      L     #LAST_BCD;
      L     #AKT_BCD; // Prüfen ob der BCD
      ==I   ;
      =     #NODIFF; // kein Unterschied in der Anwahl
      T     #LAST_BCD; // seit dem letzten Programmzyklus
NETWORK
TITLE =Verzögerungszeit BCD-WERT-Änderung bis zur Ausgangsumschaltung

      U     #DIFF;
      U     #NODIFF;
      =     L      1.0;
      BLD   103;
      CALL #TON (
           IN                       := L      1.0,
           PT                       := #DELAY,
           Q                        := #QT);

      NOP   0;
NETWORK
TITLE =

      U     #DIFF; // Wert wurde verändert
      U     #QT; // Wartezeit für Umschaltung abgelaufen
      SAVE  ; // Umschaltereignis auf ENO-AUSGANG
      SPB   SAVE; // neue Werte speichern
      BEA   ;

SAVE: L     #AKT_BCD; // Aktuelle BCD-Zahl
      T     #LAST_BCD_AKTIV; // als letzte Zahl speichern

      L     #AKT_BCD; // Aktuelle BCD-Zahl = Bit-Nr im Ausgangs-WORD
      L     1; // Eine 1 um Anzahl "BCD-Zahl" nach links schieben
      SLW   ;
      TAW   ; // Low- und High- Byte im WORD tauschen
      T     DIW [AR2,P#6.0]; // Wert an Ausgänge schreiben (Q1 bis Q9)

END_FUNCTION_BLOCK

FUNCTION_BLOCK "UP_DOWN_INT"
TITLE =UP_DOWN_INT: Wert mit Tasten vergrößeren und verkleinern
//AUTOR: Stefan Maag, Dipl.-Ing. (FH) Elektrotechnik
//DATUM: 1/2005
//
//AENDERUNGSVERMERKE:
//--------------------------------------------------------------------------------
//DATUM        NAME            AENDERUNG
//--------------------------------------------------------------------------------
//
//--------------------------------------------------------------------------------
//
//HINWEISE:
AUTHOR : 'S.Maag'
VERSION : 0.1


VAR_INPUT
  UP : BOOL ;
  DOWN : BOOL ;
  SET : BOOL ;
  SET_VALUE : INT ;
  MIN : INT ;
  MAX : INT ;
  STEP_SLOW : INT ;
  STEP_FAST : INT ;
  STEP_PULS : INT ;
  TAKT : TIME ;
  DELAY_FAST : TIME ;	//Verzögerungszeit für Umschalten auf Schnell
END_VAR
VAR_IN_OUT
  VALUE : INT ;
END_VAR
VAR
  lb_FP_UP : BOOL ;
  lb_FP_DOWN : BOOL ;
  UP_PULS : BOOL ;
  DOWN_PULS : BOOL ;
  FAST : BOOL ;
  TAKT_PULS : BOOL ;
  T1 : "TON";
  T2 : "TON";
END_VAR
BEGIN
NETWORK
TITLE =
//23.06.2012 Slow daktiviert


NETWORK
TITLE =Puls UP
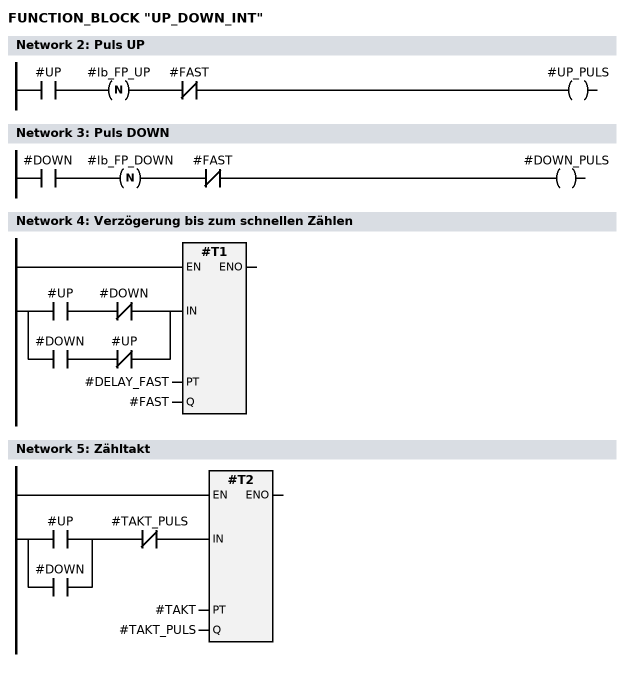

      U     #UP;
      FN    #lb_FP_UP;
      UN    #FAST;
      =     #UP_PULS;
NETWORK
TITLE =Puls DOWN

      U     #DOWN;
      FN    #lb_FP_DOWN;
      UN    #FAST;
      =     #DOWN_PULS;
NETWORK
TITLE =Verzögerung bis zum schnellen Zählen

      U(    ;
      U     #UP;
      UN    #DOWN;
      O     ;
      U     #DOWN;
      UN    #UP;
      )     ;
      =     L      0.0;
      BLD   103;
      CALL #T1 (
           IN                       := L      0.0,
           PT                       := #DELAY_FAST,
           Q                        := #FAST);

      NOP   0;
NETWORK
TITLE =Zähltakt

      U(    ;
      O     #UP;
      O     #DOWN;
      )     ;
      UN    #TAKT_PULS;
      =     L      0.0;
      BLD   103;
      CALL #T2 (
           IN                       := L      0.0,
           PT                       := #TAKT,
           Q                        := #TAKT_PULS);

      NOP   0;
NETWORK
TITLE =SET: Wert setzen

      UN    #SET;
      SPB   NE5;
      L     #SET_VALUE;
      SPA   CHK;
NE5:  NOP   0;

NETWORK
TITLE =
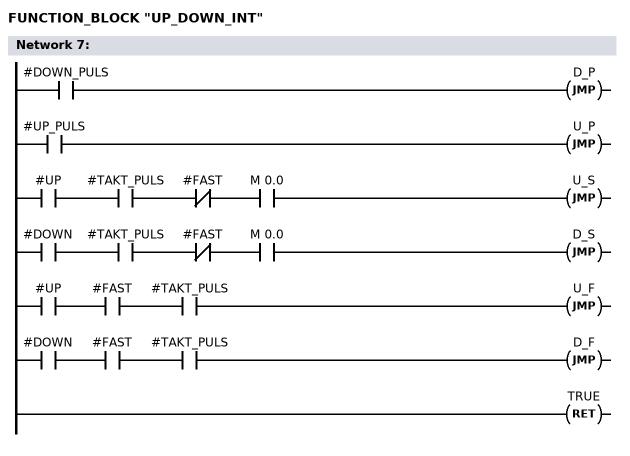

      U     #DOWN_PULS;
      SPB   D_P;

      U     #UP_PULS;
      SPB   U_P;

      U     #UP;
      U     #TAKT_PULS;
      UN    #FAST;
      U     M      0.0;
      SPB   U_S;

      U     #DOWN;
      U     #TAKT_PULS;
      UN    #FAST;
      U     M      0.0;
      SPB   D_S;

      U     #UP;
      U     #FAST;
      U     #TAKT_PULS;
      SPB   U_F;

      U     #DOWN;
      U     #FAST;
      U     #TAKT_PULS;
      SPB   D_F;
      BEA   ;

NETWORK
TITLE =

U_S:  NOP   0; // Up slow
      L     #VALUE;
      L     #STEP_SLOW;
      +I    ;
      SPA   CHK;

U_F:  NOP   0; // Up fast
      L     #VALUE;
      L     #STEP_FAST;
      +I    ;
      SPA   CHK;

U_P:  NOP   0; // Up pulse
      L     #VALUE;
      L     #STEP_PULS;
      +I    ;
      SPA   CHK;


D_S:  NOP   0; // Down slow
      L     #VALUE;
      L     #STEP_SLOW;
      -I    ;
      SPA   CHK;

D_P:  NOP   0; // Down puls
      L     #VALUE;
      L     #STEP_PULS;
      -I    ;
      SPA   CHK;

D_F:  NOP   0; // Down fast
      L     #VALUE;
      L     #STEP_FAST;
      -I    ;

CHK:  L     #MIN; // Wert auf Min/Max begrenzen
      <I    ;
      SPB   SAVE;
      TAK   ;
      L     #MAX;
      >I    ;
      SPB   SAVE;
      TAK   ;
SAVE: T     #VALUE;

END_FUNCTION_BLOCK

FUNCTION_BLOCK "m7b_SchuetzUeberwachung"
TITLE =Schützfehlerüberwachung mit Rückmeldekontakt
//AUTOR: Stefan Maag, Dipl.-Ing. (FH) Elektrotechnik
//DATUM: 12/2009
//INTERNET: www.maagic7.de
//
//AENDERUNGSVERMERKE:
//--------------------------------------------------------------------------------
//DATUM        NAME            AENDERUNG
//--------------------------------------------------------------------------------
//
//--------------------------------------------------------------------------------
//
//HINWEISE:
AUTHOR : 'S.Maag'
FAMILY : Maagic7
VERSION : 0.1


VAR_INPUT
  K : BOOL ;
  RM : BOOL ;
  IEC_TIME : TIME ;
END_VAR
VAR
  MI_TON : "TON";
END_VAR
VAR_TEMP
  XOR_RESULT : BOOL ;
  Q_TON : BOOL ;
END_VAR
BEGIN
NETWORK
TITLE =Schütz <> Rückmdlung ?

      X     #K;
      X     #RM;
      =     #XOR_RESULT;

NETWORK
TITLE =Zeitverzögerung, wenn Ansteuerung <> Rückmeldung



      U     #XOR_RESULT;
      =     L      1.0;
      BLD   103;
      CALL #MI_TON (
           IN                       := L      1.0,
           PT                       := #IEC_TIME,
           Q                        := #Q_TON);

      NOP   0;
NETWORK
TITLE =ENO-Ausgang : Fehlerausgang

      U     #Q_TON;
      SAVE  ;
      CLR   ;

END_FUNCTION_BLOCK

FUNCTION_BLOCK "POSI"
TITLE =Positionierung Achse mit Delay für Nachpositionierung bzw. Ready
//Positionierung Achse als Schrittsteuerung:
//
//Lageregelung nur während der timDelayReady.
//Soll ohne die Möglichkeit der Nachpositionierung sofort bei erreichen der
//Stopdifferenz fest abgeschaltet werden, dann timDelayReady =0
//
//
//[IN]
//FRG :       Freigabe, wenn Low, dann Abbruch der Positionierung
//SOLL:       Sollposition Achse
//IST :       Istposition Achse
//STOP_DIFF:  Vorabschaltentfernung
//TOL_POS_OK: Toleranz für Position ok Prüfung
//timDelayReady : Verzögerung für Ready (Nachpositionierung nur in dieser Zeit)
//
//[IN_OUT]
//START:      Befehl Positionierung Start, wird bei Ende oder Abbruch gelöscht
//
//[OUT]
//PLUS:       Fahrtrichtung Plus (vorw.)
//MINUS:      Fahrtrichtung Minus (rückw.)
//READY:      Positionierablauf korrekt beendet
//POS_OK:     Position innerhalb der Toleranz (ständige Prüfung)
//DSP_SNR:    Schrittnummer Positionierablauf
//
//FC_ENO:     zeigt an, dass Positionierung läuft
//
//AUTOR: Stefan Maag, Dipl.-Ing. (FH) Elektrotechnik
//DATUM: 9/2007
//
//AENDERUNGSVERMERKE:
//--------------------------------------------------------------------------------
//DATUM        NAME        AENDERUNG
//--------------------------------------------------------------------------------
//20.11.2017   S.Maag     Nachpositionierung eingeführt.
//                        timDelayReady gibt, an wie lange der Antrieb in
//                        korrekter Position sein muss, bis READY ausgegeben
//                        wird. Dann wird nicht mehr nachpositioniert.
//                        Dies ist insbesondere bei etwas instabilen Positons-
//                        erfassungen wie Laser Entfernungsmesser nötig. Sonst
//                        kann es sein, dass der Laser etwas wackelt, es wird
//                        gestoppt, die Position ist jedoch nicht im Fenster.
//--------------------------------------------------------------------------------
//
//HINWEISE:
AUTHOR : 'S.Maag'
VERSION : 0.1


VAR_INPUT
  FRG : BOOL ;	//Freigabe
  SOLL : DINT ;	//Sollwert
  IST : DINT ;	//Istwert Achse
  STOP_DIFF : DINT ;	//Vorabschaltpunkt
  TOL_POS : DINT ;	//Toleranz für Positionierung
  TOL_POS_OK : DINT ;	//Toleranz für Position ok Meldung
  timDelayReady : TIME ;
END_VAR
VAR_OUTPUT
  PLUS : BOOL ;	//Fahrtrichtung PLUS
  MINUS : BOOL ;	//Fahrtrichtung MINUS
  READY : BOOL ;	//Positionierung fertig
  POS_OK : BOOL ;	//Position innerhalb Toleranz ok
  DSP_SNR : INT ;	//Schrittnummer Positionierung, STATE
END_VAR
VAR_IN_OUT
  START : BOOL ;
END_VAR
VAR
  SNR : INT ;
  POS_DIFF : DINT ;	//aktuelle Positionsdifferenz
  FRG_GO : BOOL ;
  POS_INTERVAL : BOOL ;
  Q_TON_FRG_GO_OFF : BOOL ;
  mi_TON_FRG_GO_OFF : "TON";
END_VAR
VAR_TEMP
  tmpPosDIFF : DINT ;
  tmp_timDelay : TIME ;
END_VAR
BEGIN
NETWORK
TITLE =



NETWORK
TITLE =Zeit mindestens 1ms (da 0=RESET für IEC-Timer)

      L     L#1;
      L     #timDelayReady;
      UC    FC    21;
      T     #tmp_timDelay;

NETWORK
TITLE =Zeit Freiagbe GO ist AUS (Achse ist positioniert)

      UN    #FRG_GO;
      =     L      8.0;
      BLD   103;
      CALL #mi_TON_FRG_GO_OFF (
           IN                       := L      8.0,
           PT                       := #tmp_timDelay,
           Q                        := #Q_TON_FRG_GO_OFF);

      NOP   0;
NETWORK
TITLE =Signale Fahrtrichtung

      U(    ;
      L     #SOLL;
      L     #IST;
      -D    ;
      T     #POS_DIFF;
      UN    OV;
      SAVE  ;
      CLR   ;
      U     BIE;
      )     ;
      U     #FRG_GO;
      UN    #POS_INTERVAL;
      =     L      8.0;
      U     L      8.0;
      U     >0;
      =     #PLUS;
      U     L      8.0;
      U     <0;
      =     #MINUS;
NETWORK
TITLE =Toleranzprüfung Position

      U(    ;
      L     #POS_DIFF;
      L     L#0;
      <D    ;
      )     ;
      SPBNB _001;
      L     #POS_DIFF;
      NEGD  ;
      T     #POS_DIFF;
_001: NOP   0;
NETWORK
TITLE =Toleranzprüfung Position
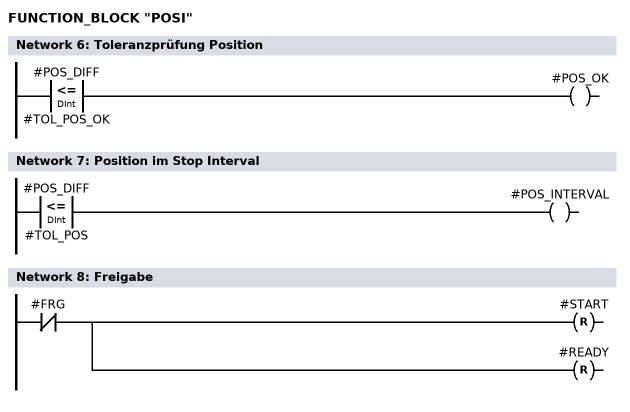

      L     #POS_DIFF;
      L     #TOL_POS_OK;
      <=D   ;
      =     #POS_OK;
NETWORK
TITLE =Position im Stop Interval

      L     #POS_DIFF;
      L     #TOL_POS;
      <=D   ;
      =     #POS_INTERVAL;
NETWORK
TITLE =Freigabe

      UN    #FRG;
      R     #START;
      R     #READY;

NETWORK
TITLE =Standard Ablaufsteuerung mit INIT und CLR-Zweig

      L     #SNR; // Schrittnummer
      SPL   CLR; // Sprungziel bei SNR>max
      SPA   INIT; // 0-Schritt, Initialisierung
      SPA   S1; // Startschritt
      SPA   S2;

CLR:  SET   ; // CLR
// hier die bei CLR zu löschenden Merker eintragen
      R     #START;
      R     #FRG_GO;

      L     1; // Schrittnummer
      T     #SNR; // auf Startschritt stellen
      T     #DSP_SNR; // Schrittnummer Anzeige
      SPA   END;

INIT: SET   ; // Initalisierung
      CLR   ;
      SPA   CLR;
      SPA   SET; // wird nur benötigt, damit die Entwicklungsumgebung die Sprungmarke nicht löscht

NETWORK
TITLE =Schrittweiterschaltung, bzw. Bausteinende

NEXT: L     #SNR; // NEXT : Schrittnummer auf nächsten
      +     1; // Schritt
SET:  T     #SNR; // Schritt setzten

END:  L     #SNR; // Sprungmarke für Baustein ENDE
      T     #DSP_SNR; // Schrittnummer Anzeige
      L     1; // Wenn Ablauf läuft, dann ENO-Ausgang = 1
      >I    ;
      SAVE  ;
      CLR   ;
      BEA   ;

NETWORK
TITLE =Positionierung START?
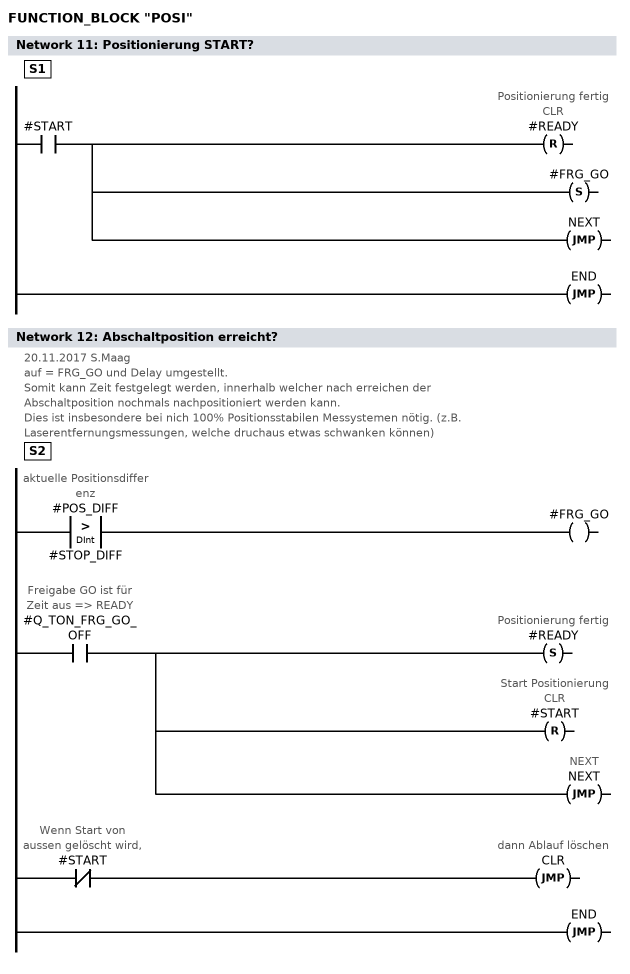

S1:   U     #START;
      R     #READY; // Positionierung fertig CLR
      S     #FRG_GO;
      SPB   NEXT;
      SPA   END;

NETWORK
TITLE =Abschaltposition erreicht?
//20.11.2017 S.Maag
//auf = FRG_GO und Delay umgestellt.
//Somit kann Zeit festgelegt werden, innerhalb welcher nach erreichen der
//Abschaltposition nochmals nachpositioniert werden kann.
//Dies ist insbesondere bei nich 100% Positionsstabilen Messystemen nötig. (z.B.
//Laserentfernungsmessungen, welche druchaus etwas schwanken können)
S2:   NOP   0;
      L     #POS_DIFF; // aktuelle Positionsdifferenz
      L     #STOP_DIFF; // Vorabschaltpunkt
      >D    ;
      =     #FRG_GO;

      U     #Q_TON_FRG_GO_OFF; // Freigabe GO ist für Zeit aus => READY
      S     #READY; // Positionierung fertig
      R     #START; // Start Positionierung CLR
      SPB   NEXT; // NEXT

      UN    #START; // Wenn Start von aussen gelöscht wird,
      SPB   CLR; // dann Ablauf löschen
      SPA   END;


END_FUNCTION_BLOCK

FUNCTION_BLOCK "m7b_FU_RFR"
TITLE =Reglerfreigabe mit Nachlauf aus vw/rw Signal erzeugen
//AUTOR: Stefan Maag, Dipl.-Ing. (FH) Elektrotechnik
//DATUM: 01/2013
//INTERNET: www.maagic7.de
//
//AENDERUNGSVERMERKE:
//--------------------------------------------------------------------------------
//DATUM        NAME         AENDERUNG
//--------------------------------------------------------------------------------
//13.06.2020   S.Maag       in Library aufgenommen
//--------------------------------------------------------------------------------
//
//HINWEISE:
AUTHOR : 'S.Maag'
VERSION : 0.1


VAR_INPUT
  vw : BOOL ;	//vorwärts
  rw : BOOL ;	//rückwärts
  FRG : BOOL ;
  timTON_MSG : TIME ;	//Verzögerung Meldung RFR
  timTOF_RFR : TIME ;	//Nachlauf Reglerfreigabe
END_VAR
VAR_OUTPUT
  RFR : BOOL ;	//Ausgang Reglerfreigabe FU
  MSG_RFR : BOOL ;	//Meldung verzögert Reglerfreigabe o.k.
END_VAR
VAR
  Q_TON_MSG : BOOL ;
  Q_TOF_RFR : BOOL ;
  TOF_RFR : "TOF";
  TON_MSG : "TON";
END_VAR
VAR_TEMP
  xTON_MSG_IS_ZERO : BOOL ;
  xTOF_RFR_IS_ZERO : BOOL ;
END_VAR
BEGIN
NETWORK
TITLE =



NETWORK
TITLE =Verzögerungszeit Meldung ist 0 ms
//bei 0ms starten IEC Timer nicht und Ausgang bleibt immer lo,
//Aufruf mit 0ms ist RESET
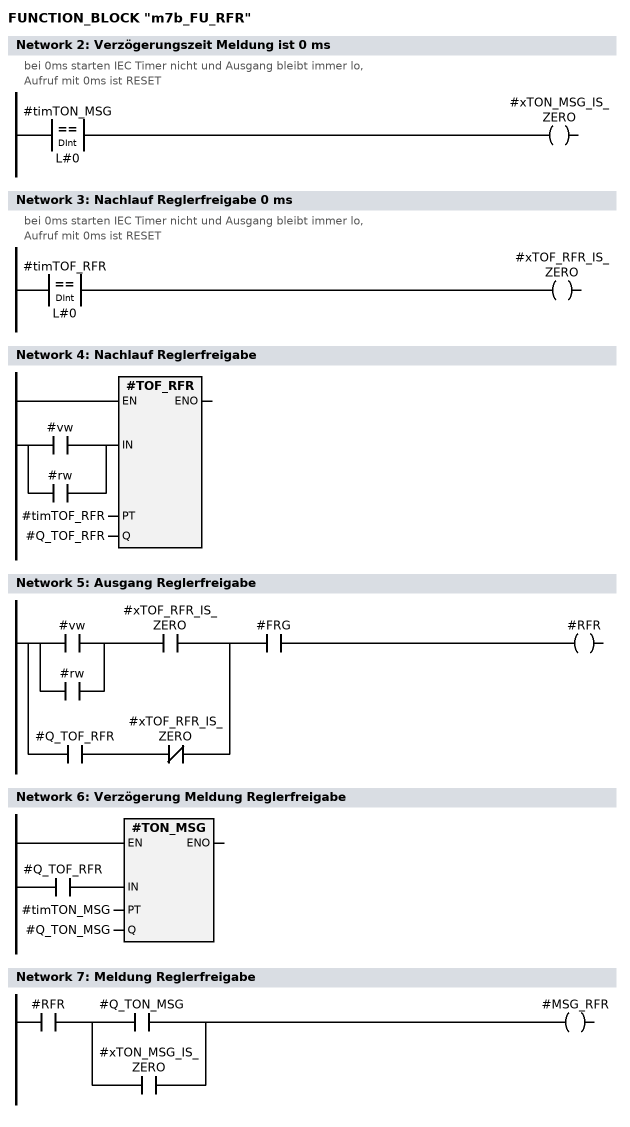
      L     #timTON_MSG;
      L     L#0;
      ==D   ;
      =     #xTON_MSG_IS_ZERO;
NETWORK
TITLE =Nachlauf Reglerfreigabe 0 ms
//bei 0ms starten IEC Timer nicht und Ausgang bleibt immer lo,
//Aufruf mit 0ms ist RESET
      L     #timTOF_RFR;
      L     L#0;
      ==D   ;
      =     #xTOF_RFR_IS_ZERO;
NETWORK
TITLE =Nachlauf Reglerfreigabe

      U(    ;
      O     #vw;
      O     #rw;
      )     ;
      =     L      1.0;
      BLD   103;
      CALL #TOF_RFR (
           IN                       := L      1.0,
           PT                       := #timTOF_RFR,
           Q                        := #Q_TOF_RFR);

      NOP   0;
NETWORK
TITLE =Ausgang Reglerfreigabe

      U(    ;
      U(    ;
      O     #vw;
      O     #rw;
      )     ;
      U     #xTOF_RFR_IS_ZERO;
      O     ;
      U     #Q_TOF_RFR;
      UN    #xTOF_RFR_IS_ZERO;
      )     ;
      U     #FRG;
      =     #RFR;
NETWORK
TITLE =Verzögerung Meldung Reglerfreigabe



      U     #Q_TOF_RFR;
      =     L      1.0;
      BLD   103;
      CALL #TON_MSG (
           IN                       := L      1.0,
           PT                       := #timTON_MSG,
           Q                        := #Q_TON_MSG);

      NOP   0;
NETWORK
TITLE =Meldung Reglerfreigabe

      U     #RFR;
      U(    ;
      O     #Q_TON_MSG;
      O     #xTON_MSG_IS_ZERO;
      )     ;
      =     #MSG_RFR;
END_FUNCTION_BLOCK

FUNCTION_BLOCK "m7b_HydraulicPump"
TITLE =Steuerung Hydraulik mit Lastventil : Hydraulic with load valve
//Steuerung Hydraulikpumpe mit Lastventil!
//
//Einstellbare Nachlaufzeit für Hydraulikpumpe.
//Durch einstellbare Vor- und Nachlaufzeit für Lastventil (Meldung Druck auf
//Hydraulik), verwendbar auch für Hydrauliken mit Porportionalventilen. Bei
//Proportinalsteuerung muss das Lastventil mindestens so lange nachlaufen, wie
//die
//längste Rampenzeit der Ventile. Durch die Vorlaufzeit des Lastventils kann man
//sicherstellen, dass auf jeden Fall Druck ansteht, bevor man die
//Proportionalventile ansteuert.
//
//[IN]
//START        : Befehl, Hydraulik starten
//FRG          : Freigabe für Hydraulik (Netz_ok, Motorschutz usw. verschalten)
//T_HYDR_OFF   : Nachlaufzeit Hydraulikpumpe IEC-Time-Format
//T_Y_LOAD_OFF : Nachlaufzeit Lastventil (> max. Rampenzeiten bei Prop.Ventilen)
//T_MSG_LOAD_ON: Verzögerung Meldung Lastventil ein (Vorlauf Lastventil)
//
//[OUT]
//PUMP          : Ausgang Hydraulikpumpe EIN
//Y_LOAD        : Ausgang Lastventil
//MSG_PUMP_READY: Meldung Hydraulik bereit (=durchgeschleiftes Singal FRG)
//MSG_PUMP_RUN  : Meldung Hydraulikpumpe läuft (fix verzögert 500ms)
//MSG_LOAD_ON   : Meldung Lastventil ist ein (Druck auf Hydraulik) - verzögert
//
//AUTOR: Stefan Maag, Dipl.-Ing. (FH) Elektrotechnik
//DATUM: 11/2008
//INTERNET: www.maagic7.de
//
//AENDERUNGSVERMERKE:
//--------------------------------------------------------------------------------
//DATUM        NAME            AENDERUNG
//--------------------------------------------------------------------------------
//17.09.2010  S.Maag      Reset der iecZeit TOF_HydrPump über 0 im den Zeitwert
//                        damit läuft Pumpe nach Freigabeverlust nicht wieder an
//--------------------------------------------------------------------------------
//
//HINWEISE:
AUTHOR : 'S.Maag'
FAMILY : Maagic7
VERSION : 0.1


VAR_INPUT
  START : BOOL ;	//Hydraulik START
  FRG : BOOL ;	//Freigabe Hydraulikpumpe
  T_HYDR_OFF : TIME ;	//Nachlaufzeit Hydraulikpumpe
  T_Y_LOAD_OFF : TIME ;	//Nachlauf Lastventil
  T_MSG_LOAD_ON : TIME ;
END_VAR
VAR_OUTPUT
  PUMP : BOOL ;	//Ausgang Hydraulikpumpe EIN
  Y_LOAD : BOOL ;	//Ausgang Lastventil
  MSG_PUMP_READY : BOOL ;	//Meldung Hydraulik bereit
  MSG_PUMP_RUN : BOOL ;	//Meldung Hydraulik läuft
  MSG_LOAD_ON : BOOL ;	//Meldung Lastventil ein
END_VAR
VAR
  Q_T_Hydraulic : BOOL ;
  Q_PUMP : BOOL ;
  Q_LOAD_REQ : BOOL ;
  Q_T_LOAD : BOOL ;
  Q_LOAD : BOOL ;
  TOF_HydrPump : "TOF";
  TON_MSG_RUN : "TON";
  TON_LOAD_ON : "TON";
  TOF_LOAD : "TOF";
END_VAR
VAR_TEMP
  DSP_TIME : TIME ;
  m_T_HYDR_OFF : TIME ;
END_VAR
BEGIN
NETWORK
TITLE =



NETWORK
TITLE =Zeit Hydraulik aus auf temporären Zwischenspeicher
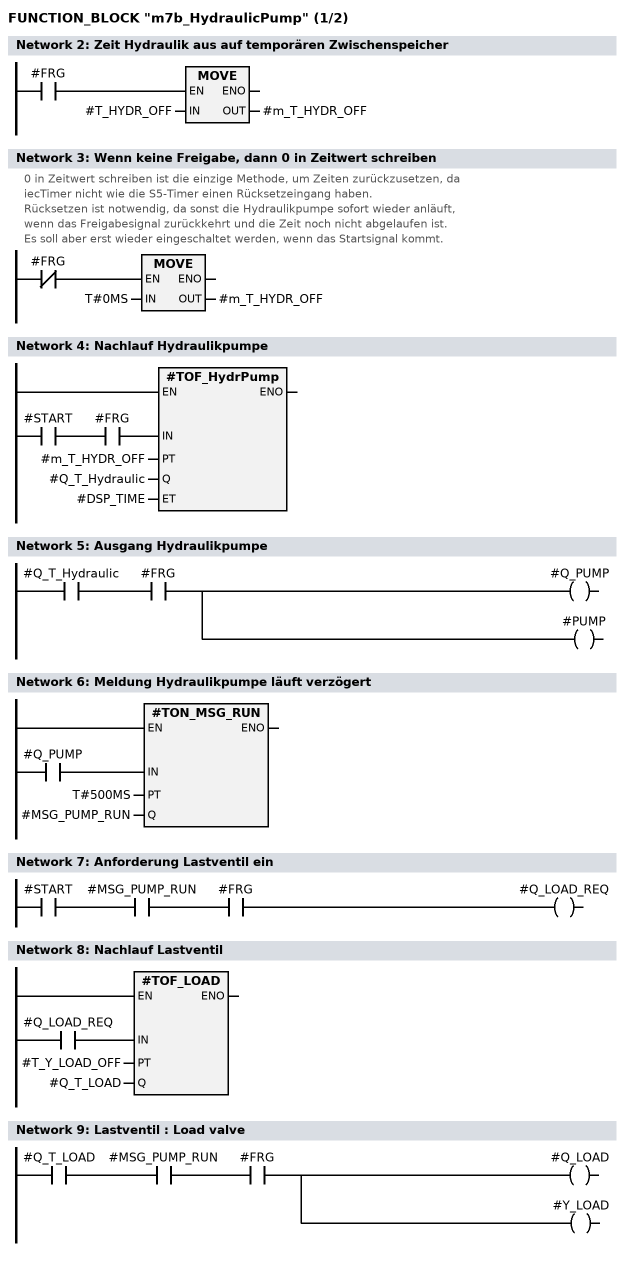

      U     #FRG;
      SPBNB _001;
      L     #T_HYDR_OFF;
      T     #m_T_HYDR_OFF;
_001: NOP   0;
NETWORK
TITLE =Wenn keine Freigabe, dann 0 in Zeitwert schreiben
//0 in Zeitwert schreiben ist die einzige Methode, um Zeiten zurückzusetzen, da
//iecTimer nicht wie die S5-Timer einen Rücksetzeingang haben.
//
//Rücksetzen ist notwendig, da sonst die Hydraulikpumpe sofort wieder anläuft,
//wenn das Freigabesignal zurückkehrt und die Zeit noch nicht abgelaufen ist.
//Es soll aber erst wieder eingeschaltet werden, wenn das Startsignal kommt.
//
      UN    #FRG;
      SPBNB _002;
      L     T#0MS;
      T     #m_T_HYDR_OFF;
_002: NOP   0;
NETWORK
TITLE =Nachlauf Hydraulikpumpe



      U     #START;
      U     #FRG;
      =     L      8.0;
      BLD   103;
      CALL #TOF_HydrPump (
           IN                       := L      8.0,
           PT                       := #m_T_HYDR_OFF,
           Q                        := #Q_T_Hydraulic,
           ET                       := #DSP_TIME);
      NOP   0;
NETWORK
TITLE =Ausgang Hydraulikpumpe

      U     #Q_T_Hydraulic;
      U     #FRG;
      =     #Q_PUMP;
      =     #PUMP;
NETWORK
TITLE =Meldung Hydraulikpumpe läuft verzögert

      U     #Q_PUMP;
      =     L      8.0;
      BLD   103;
      CALL #TON_MSG_RUN (
           IN                       := L      8.0,
           PT                       := T#500MS,
           Q                        := #MSG_PUMP_RUN);

      NOP   0;
NETWORK
TITLE =Anforderung Lastventil ein

      U     #START;
      U     #MSG_PUMP_RUN;
      U     #FRG;
      =     #Q_LOAD_REQ;
NETWORK
TITLE =Nachlauf Lastventil

      U     #Q_LOAD_REQ;
      =     L      8.0;
      BLD   103;
      CALL #TOF_LOAD (
           IN                       := L      8.0,
           PT                       := #T_Y_LOAD_OFF,
           Q                        := #Q_T_LOAD);

      NOP   0;
NETWORK
TITLE =Lastventil : Load valve

      U     #Q_T_LOAD;
      U     #MSG_PUMP_RUN;
      U     #FRG;
      =     #Q_LOAD;
      =     #Y_LOAD;
NETWORK
TITLE =Meldung Lastventil ein : Message Load valve on
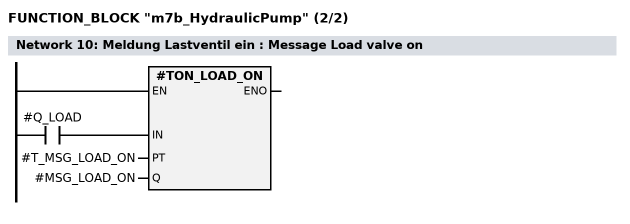

      U     #Q_LOAD;
      =     L      8.0;
      BLD   103;
      CALL #TON_LOAD_ON (
           IN                       := L      8.0,
           PT                       := #T_MSG_LOAD_ON,
           Q                        := #MSG_LOAD_ON);

      NOP   0;
NETWORK
TITLE =ENO-Ausgang = Lastventil

      U     #Q_LOAD;
      SAVE  ;
      CLR   ;

END_FUNCTION_BLOCK

FUNCTION_BLOCK "m7b_ZylSensorCtrl"
TITLE =ZylinderSensorControl, für Zylinder mit 2 Sensoren
//Dier FB erledigt 2 Funktionen
//1. Verzögerung der Zylindersensoren und generieren der Positionsmeldungen
//2. Überwachung der Zylinderbewegungen anhand der max. erlaubten Bewegungszeit
//   bis der entsprechende Positionssensor belegt ist.
//
//Wird in der angebenen Zeit die Zylinderendstellung nicht erreicht, so wird
//ERROR für die entsprechende Richtung ausgegeben. Der ENO-Ausgang des FC erhält
//den ODER-verknüpten Error-Zustand. Ist also bei Fehler, egal welcher Richtung
//High
//
//Auf die SFBs TON, TOF wird verzichtet, da diese bereits je 22Byte an statischen
//Daten verbrauchen. Dies wurde hauptsächlich wegen Speicherproblemen bei den
//kleinen CPUs (312/313) so ausgeführt.
//
//AUTOR: Stefan Maag, Dipl.-Ing. (FH) Elektrotechnik
//DATUM: 3/2008
//INTERNET: www.maagic7.de
//
//HINWEISE: Entstand aus FC7: m7ZylinderFehlerEx
//
//AENDERUNGSVERMERKE:
//--------------------------------------------------------------------------------
//DATUM        NAME            AENDERUNG
//--------------------------------------------------------------------------------
//03/12/2013   S.Maag      SFC64 TimeTick Zeitdifferenz korrigiert
//                         da 31Bit, Fehler bei Überlauf.
//                         UC FC256 "ABS_DIFF_S7SysTime" verwendet
//--------------------------------------------------------------------------------
//
AUTHOR : 'S.Maag'
FAMILY : Maagic7
VERSION : 0.1


VAR_INPUT
  SENS_GST : BOOL ;	//Sensor Grundstellung
  SENS_AST : BOOL ;	//Sensor Arbeitsstellung
  Y_GST : BOOL ;	//Eingang Schaltsignal Grundstellungs-Ventil
  Y_AST : BOOL ;	//Eingang Schaltsignal Arbeitsstellungs-Ventil
  iec_T_Err : TIME ;	//Zeit für Bewegung Fehlerüberwachung, IEC-Format
  iec_T_PosDelay : TIME ;	//Verzögerungszeit für Positionssensoren
END_VAR
VAR_OUTPUT
  POS_GST : BOOL ;	//Position Grundstellung
  POS_AST : BOOL ;	//Position Arbeitsstellung
  ERR_GST : BOOL ;	//Ausgang Fehler Sensor Grundstellung
  ERR_AST : BOOL ;	//Ausgang Fehler Sensor Arbeitsstellung
  STATUS : INT ;	//0=zu 1=auf 2=fährt 3=Fehler zu  4=Fehler auf
END_VAR
VAR
  FP_YGST : BOOL ;	//Flanke positiv Ventil Grundstellung
  FP_YAST : BOOL ;	//Flanke positiv Ventil Arbeitsstellung
  FP_B_GST : BOOL ;
  FP_B_AST : BOOL ;
  aktSysTime : TIME ;
  T_FP_B_GST : TIME ;	//akt. SysZeit Sensor GST Flanke
  T_FP_B_AST : TIME ;	//akt. SysZeit Sensor AST Flanke
  tmpErrTime : TIME ;	//Speichervariable für Zeit
END_VAR
BEGIN
NETWORK
TITLE =aktuelle Systemzeit Zwischenspeichern

      CALL "TIME_TCK" (// aktuelle Systemzeit auslesen
           RET_VAL                  := #aktSysTime);
      NOP   0;
NETWORK
TITLE =Systemzeit bei Sensor Grundstellung belegt
//Zeit bei der Sensor belegt wurde.
      U     #SENS_GST;
      FP    #FP_B_GST;
      SPBNB _001;
      L     #aktSysTime;
      T     #T_FP_B_GST;
_001: NOP   0;
NETWORK
TITLE =Systemzeit bei Sensor Arbeitsstellung belegt
//Zeit bei der Sensor belegt wurde.
      U     #SENS_AST;
      FP    #FP_B_AST;
      SPBNB _002;
      L     #aktSysTime;
      T     #T_FP_B_AST;
_002: NOP   0;
NETWORK
TITLE =Ausgang Position Grundstellung erreicht
//Verzögerung Position Grundstellung
      UN    #SENS_GST; // Sensor Grundstellung nicht aktiv
      R     #POS_GST; // dann Position Grundstellung clr
      SPB   ne4; // Netzwerkende
      L     #aktSysTime; // Wenn Grundstellungssensor High, dann
      L     #T_FP_B_GST; // Zeit überpüfen wie lange bereits
      UC    "m7b_ABS_DIFF_S7SysTime"; // Zeitdifferenz absolut ermitteln
      L     #iec_T_PosDelay; // Wenn größer als Verzögerung,
      >=D   ;
      S     #POS_GST; // dann Position Grundstellung setzen
ne4:  NOP   0;

NETWORK
TITLE =Ausgang Position Arbeitsstellung erreicht
//Verzögerung Position Arbeitsstellung
      UN    #SENS_AST; // Sensor Arbeitsstellung nicht aktiv
      R     #POS_AST; // dann Position Arbeitsstellung clr
      SPB   ne5; // Netzwerkende
      L     #aktSysTime; // Wenn Arbeitsstellungssensor High, dann
      L     #T_FP_B_AST; // Zeit überpüfen wie lange bereits
      UC    "m7b_ABS_DIFF_S7SysTime"; // Zeitdifferenz absolut ermitteln
      L     #iec_T_PosDelay; // Wenn größer als Verzögerung,
      >=D   ;
      S     #POS_AST; // dann Position Arbeitsstellung setzen
ne5:  NOP   0;

NETWORK
TITLE =Zeit bei Bewegung Start speichern

      U     #Y_GST; // falls beide Ventile gleichzeitg angesteuert sind
      U     #Y_AST; // dann Zeitüberwachung solange starten bis ein
      SPB   SVT; // Ventil abgeschaltet wird. Erst dann ist def. Zustand

      U     #Y_GST; // Ventil Grundstellung
      FP    #FP_YGST; // Flanke Ventilansteuerung
      SPB   SVT; // Save Time

      U     #Y_AST; // Ventil Arbeitsstellung
      FP    #FP_YAST; // Flanke Ventilansteuerung
      SPB   SVT; // Save Time

      SPA   NE1;

SVT:  NOP   0; // Zeit bei Bewegung Start speichern
      CALL "TIME_TCK" (// Systemzeit wird zur Bewegungsüberwachung verwendet
           RET_VAL                  := #tmpErrTime);// dadurch erspart man sich Timerübergaben

NE1:  NOP   0;
NETWORK
TITLE =Prüfen, ob beide Sensoren belegt sind => Fehler

      U     #SENS_GST;
      U     #SENS_AST;
      SPBN  NE2;
      =     #ERR_GST;
      =     #ERR_AST;
      SAVE  ;
      BEA   ;
NE2:  NOP   0;

NETWORK
TITLE =Zeit überprüfen, ob Endstellung erreicht ist

      U     #Y_GST; // Ventil Grundstellung
      UN    #SENS_GST; // Sensor GST nicht erreicht
      SPB   TCHK; // Prüfen ob max. Zeit Abgelaufen

      U     #Y_AST; // Ventil Arbeitsstellung
      UN    #SENS_AST; // Sensor Arbeitsstellung nicht erreicht
      SPB   TCHK; // Prüfen ob max. Zeit Abgelaufen

      CLR   ;
      =     #ERR_GST;
      =     #ERR_AST;
      SAVE  ;
      SPA   NE8; // Netzwerkende

TCHK: NOP   0; // Zeit Abgelaufen?
      L     #aktSysTime;
      L     #tmpErrTime; // Zeit bei Start Bewegung
      UC    "m7b_ABS_DIFF_S7SysTime";
      L     #iec_T_Err; // Zeit für Bewegung
      >D    ; // Zeit abgelaufen
      SAVE  ; // Fehler im BIE-Bit speichern
      CLR   ;

      U     BIE;
      U     #Y_GST; // Ventil Grundstellung angesteuert, dann
      =     #ERR_GST; // Fehler Sensor Grundstellung

      U     BIE; // gespeicherter Fehlerzustand im BIE-Bit
      U     #Y_AST; // und Ventil Arbeitsstellung, dann
      =     #ERR_AST; // Fehler Sensor Arbeitsstellung
NE8:  NOP   0;
NETWORK
TITLE =Statusanzeige bearbeiten
//0 = geschlossen
//1 = offen
//2 = fährt
//3 = Störung bei zu
//4 = Störung bei auf
      L     3; // Fehler zu
      U     #ERR_GST;
      SPB   SAVE;

      L     4; // Fehler auf
      U     #ERR_AST;
      SPB   SAVE;

      L     0; // zu
      U     #POS_GST;
      SPB   SAVE;

      L     1; // offen
      U     #POS_AST;
      SPB   SAVE;

      L     2; // fährt

SAVE: T     #STATUS;
      SET   ;
      SAVE  ;
      CLR   ;

END_FUNCTION_BLOCK

FUNCTION_BLOCK "m7b_DISTANCE_COUNTER"
TITLE =Weg-Zähler (km Zähler)
//Dieser FB arbeitet als Weg-Zähler, vergleichbar einem km-Zähler.
//
//IN: ENDODER: Positionswert des zu zählenden Encoders
//IN: INKR   : Anzahl der Weginkremente, die jeweils eine Zähleinheit bilden
//IN: FRG    : Zählfreigabe; Zählvorgang an der akt. EncoderPos. beginnen
//IN: RICHTUNG: hiermit kann die Zählrichtung für den Weg angebeben werden 0:+/1:-
//
//Der Baustein verfügt über eine integrierte Fehlerkorrektur: D.h. es soll z.B.
//in einer Teilung von je 100 INKR gezählt werden. Dabei kommt es vor, bedingt
//durch SPS Zykluszeit usw., das das Zählerereignis erst bei einem Weg von z.B.
//105 INKR bearbeitet wird. Dies wird korrigiert, indem beim nächsten Mal die
//Soll-Inkremente dann auf 95 festgelegt werden usw. Dies verhindert einen sich
//aufschaukelden Fehler!
//
//AUTOR: Stefan Maag, Dipl.-Ing. (FH) Elektrotechnik
//DATUM: 3/2003
//INTERNET: www.maagic7.de
//
//AENDERUNGSVERMERKE:
//--------------------------------------------------------------------------------
//DATUM        NAME            AENDERUNG
//--------------------------------------------------------------------------------
//05.05.2010   S.Maag          von FC auf FB umgestellt, Code unverändert
//--------------------------------------------------------------------------------
//
//HINWEISE:
AUTHOR : 'S.Maag'
FAMILY : Maagic7
VERSION : 0.1


VAR_INPUT
  ENCODER : DINT ;	//Positionswert Encoder
  INKR : DINT ;	//Inkremente für einen gezählten Wegimpuls (TEILUNG)
  FRG : BOOL ;	//Zählfreigabe
  RICHTUNG : BOOL ;	//Zählrichtung 0 = vorw. / 1 = rückw.
END_VAR
VAR_OUTPUT
  Overflow : BOOL ;	//Overflow +
  Underflow : BOOL ;	//Overflow - (underflow)
END_VAR
VAR_IN_OUT
  Weg : DINT ;	//Speicher für Wegwert
END_VAR
VAR
  memWeg : DINT ;	//Hilfsspeicher für Zwischenspeicherung Startwert Zählen
  memINKR : DINT ;
  bStart : BOOL ;	//Hilfsmerker Zähler gestartet
END_VAR
BEGIN
NETWORK
TITLE =Satusausgänge Zählung löschen, werden im Code 1malig gesetzt

      CLR   ; // ENO-Ausgang löschen
      SAVE  ; // bei Zählereignis 1x gesetzt
      =     #Overflow; // Überlauf positiv
      =     #Underflow; // Überlauf negativ

NETWORK
TITLE =


      UN    #FRG; // keine FRG
      R     #bStart; // Zähler gestartet clr
      BEB   ;

NETWORK
TITLE =Zähler starten: jedesmal bei Wiederkehr von FRG neu starten

      U     #bStart; // Zähler bereits gestartet
      SPB   NWE; // Netzwerkende

      S     #bStart; // Zähler ist gestartet

      L     #ENCODER; // Encoder-Wert
      T     #memWeg; // als Startwert speichern

      L     #INKR; // Anzahl der zu zählenden Inkremente
      T     #memINKR; // in mem-Varible speichern

NWE:  NOP   0;
NETWORK
TITLE =
//Statubsbits: A0 (<0) : A1 (>0)
//Statusbist bei
//positivem Überlauf (Overflow) : OV, A0 = 1
//negativem Überlauf (Underflow): OV, 1  = 1
      L     #ENCODER; // aktueller Encoder Wert
      L     #memWeg; // Hilfsspeicher StartWert Encoder
      -D    ; // zurückgelegte Strecke
      SPP   weit; // Wenn positiv dann weiter
      NEGD  ; // Vorzeichen drehen
weit: L     #memINKR; // Anzahl der Inkremente pro Wegeinheit
      -D    ; // >=0 : Wegeinheit erreicht; >0 zuviel gez. INKR
      SPPZ  cnt; // springe zu zählen, wenn >=0
      BEA   ;

cnt:  L     #INKR; // Inkremente pro Wegeinheit
      TAK   ; // zu viel gezählte INKR in Akku 1 zurück
      -D    ; // Korrektur SollInkr.: beim nächsten mal weniger zählen
      SPMZ  nsav; // Wenn Ergebnis <=0, dann nicht speichern (Encoderüberlauf)
      T     #memINKR; // beim nächsten mal zu zählende Inkremente

nsav: L     1;
      UN    #RICHTUNG; // keine Richtungsumkehr
      SPB   inc; // Weg erhöhen
      NEGD  ; // Vorzeichen drehen
inc:  L     #Weg;
      +D    ;
      T     #Weg;

      L     #ENCODER; // Encoder-Wert
      T     #memWeg; // als Startwert speichern

      SET   ; // ENO-Ausgang bei jedem Zählereignis 1x aktivieren
      SAVE  ;
      CLR   ;

      UN    OV; // Überlaufbit
      BEB   ; // Wenn kein Überlauf, dann Ende

      U     <0; // Abfrage Statusbit A0 (Wert im Akku <0)
      =     #Overflow; // Overfolw +, wenn von +2147483647 auf -2147483648 wechselt

      U     >0; // Abfrage Statusbit A1 (Wert im Akku >0)
      =     #Underflow; // Underflow -, wenn von -2147483648 auf +2147483647 wechselt


END_FUNCTION_BLOCK

FUNCTION_BLOCK "m7b_MotorLoadControl"
TITLE =Unter- Überlast- Auswertung Motor
//AUTOR: Stefan Maag, Dipl.-Ing. (FH) Elektrotechnik
//DATUM: 4/2012
//
//
//AENDERUNGSVERMERKE:
//--------------------------------------------------------------------------------
//DATUM        NAME        AENDERUNG
//--------------------------------------------------------------------------------
//05.04.2020   S.Maag      Anordung der Ein- / Ausgänge optimiert und
//                         Bezeichnungsschema auf Stanard:
//                         MinMin, Min, Max, MaxMax geändert.
//                         In Library aufgenommen
//--------------------------------------------------------------------------------
//
//HINWEISE:
AUTHOR : 'S.Maag'
FAMILY : Maagic7
VERSION : 2.0


VAR_INPUT
  StartUp : BOOL ;	//Motor StartUp is active
  RUN : BOOL ;	//Motor RUN message
  EXT_Inhibit : BOOL ;	//External inibit (externes Sperrsignal)
  iMaxMax : INT  := 1200;	//Level MaxMax
  iMax : INT  := 1100;	//Level Max
  iMin : INT  := 800;	//Level Min
  iMinMin : INT  := 700;	//Level MinMIn
  iMotor_IorP : INT ;	//Motor actual current or power
  iNominal_IorP : INT ;	//Nominal Motor current or power
  tim_MaxMax : TIME ;	//Delay for MaxMax Error
  tim_MinMin : TIME ;	//Delay for MinMin Error
  RESET : BOOL ;
END_VAR
VAR_OUTPUT
  ERR_MaxMax : BOOL ;	//Error MaxMax, delayed (Overload Error) - must be RESET
  MSG_MaxMax : BOOL ;	//Message MaxMax, undelayed (Overload)
  MSG_Max : BOOL ;	//Message Max, undelayed (Overload warning)
  MSG_OK : BOOL ;	//Message ok. (Load ok.)0
  MSG_Min : BOOL ;	//Message Min, undelayed (Underload warning)
  MSG_MinMin : BOOL ;	//Message MinMin, undelayed (Underload)
  ERR_MinMin : BOOL ;	//Error MinMin, delayed (Underlaod Error) - must be RESET
  iMotorLoad : INT ;	//Displays the MotorLoad [%] [0..100..]
  iStatus : INT ;	//HMI Status
END_VAR
VAR
  TON_MinMin : "TON";
  TON_MaxMax : "TON";
END_VAR
VAR_TEMP
  HM_MSG_MaxMax : BOOL ;
  HM_MSG_MinMin : BOOL ;
  Q_TON_MaxMax : BOOL ;
  Q_TON_MinMin : BOOL ;
  DSP_TIME : TIME ;
  tmpMotorLoad : INT ;
END_VAR
BEGIN
NETWORK
TITLE =



NETWORK
TITLE =Calulate the Motor load in percent [%],[0..100]
//calculate as DINT to be sure not exceeding the INT Range
      L     #iMotor_IorP; // actual Motor current or power
      ITD   ;
      L     L#100; // %-Range
      *D    ;
      L     #iNominal_IorP; // Nominal Motor current or power
      ITD   ;
      /D    ;
      T     #tmpMotorLoad; // Motor load % 0..100
      T     #iMotorLoad;
NETWORK
TITLE =Oveerload analysis / Ueberlastauswertung
//======================================================================
//                     O V E R L O A D
//======================================================================


NETWORK
TITLE =MaxMax Overload
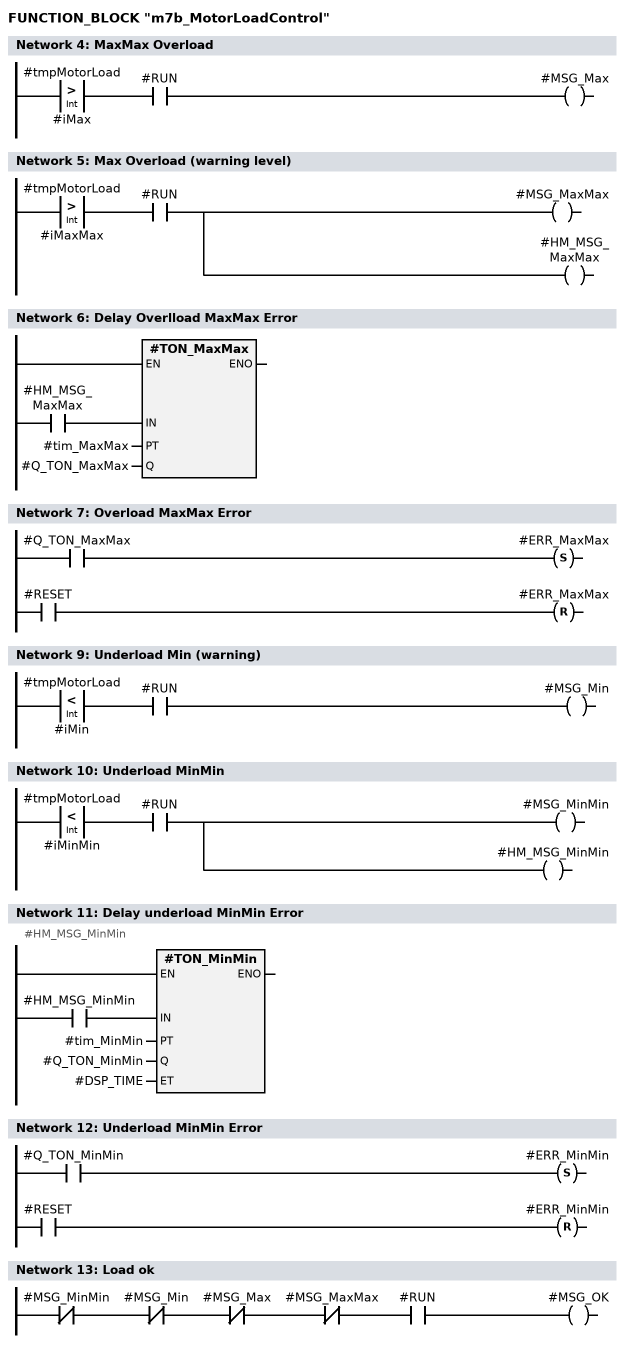

      U(    ;
      L     #tmpMotorLoad;
      L     #iMax;
      >I    ;
      )     ;
      U     #RUN;
      =     #MSG_Max;
NETWORK
TITLE =Max Overload (warning level)

      U(    ;
      L     #tmpMotorLoad;
      L     #iMaxMax;
      >I    ;
      )     ;
      U     #RUN;
      =     #MSG_MaxMax;
      =     #HM_MSG_MaxMax;
NETWORK
TITLE =Delay Overlload MaxMax Error

      U     #HM_MSG_MaxMax;
      =     L      8.0;
      BLD   103;
      CALL #TON_MaxMax (
           IN                       := L      8.0,
           PT                       := #tim_MaxMax,
           Q                        := #Q_TON_MaxMax);

      NOP   0;
NETWORK
TITLE =Overload MaxMax Error

      U     #Q_TON_MaxMax;
      S     #ERR_MaxMax;
      U     #RESET;
      R     #ERR_MaxMax;
      NOP   0;
NETWORK
TITLE =Underload analysis / Unterlastauswertung
//======================================================================
//                   U N D E R L O A D
//======================================================================


NETWORK
TITLE =Underload Min (warning)



      U(    ;
      L     #tmpMotorLoad;
      L     #iMin;
      <I    ;
      )     ;
      U     #RUN;
      =     #MSG_Min;
NETWORK
TITLE =Underload MinMin

      U(    ;
      L     #tmpMotorLoad;
      L     #iMinMin;
      <I    ;
      )     ;
      U     #RUN;
      =     #MSG_MinMin;
      =     #HM_MSG_MinMin;
NETWORK
TITLE =Delay underload MinMin Error
//#HM_MSG_MinMin
      U     #HM_MSG_MinMin;
      =     L      8.0;
      BLD   103;
      CALL #TON_MinMin (
           IN                       := L      8.0,
           PT                       := #tim_MinMin,
           Q                        := #Q_TON_MinMin,
           ET                       := #DSP_TIME);
      NOP   0;
NETWORK
TITLE =Underload MinMin Error

      U     #Q_TON_MinMin;
      S     #ERR_MinMin;
      U     #RESET;
      R     #ERR_MinMin;
      NOP   0;
NETWORK
TITLE =Load ok

      UN    #MSG_MinMin;
      UN    #MSG_Min;
      UN    #MSG_Max;
      UN    #MSG_MaxMax;
      U     #RUN;
      =     #MSG_OK;
NETWORK
TITLE =Display status
//======================================================================
//                       S T A T U S
//======================================================================


NETWORK
TITLE =Display Status
//0 : OFF
//1 : MSG MinMin    (Unterlast)
//2 : MSG Min       (Unterlast Warnung)
//3 : MSG ok.       (Last o.k.)
//4 : MSG_Max       (Überlast Warnung)
//5 : MSG_MaxMax    (Überlast)
//6 : Error MaxMax  (Überlast Störung)
//7 : Error MinMin  (Unterlast Störung)
//8 : External inhibit
//
//Überlast- und Unterlast- Error müssen im Status-Wert nebeneinander liegen, somit
//kann man anhand dieses Wertes in WinCC eine Reset-Schaltfläche einblenden
      L     6;
      U     #ERR_MaxMax; // Überlast Error
      SPB   save;

      L     7;
      U     #ERR_MinMin; // Unterlast Error
      SPB   save;


      L     5;
      U     #MSG_MaxMax; // Überlast
      SPB   save;

      L     4;
      U     #MSG_Max; // Überlast Alarm
      SPB   save;

      L     3; // Last o.k.
      U     #MSG_OK;
      SPB   save;

      L     1; // Unterlast
      U     #HM_MSG_MinMin; // muss vor UL Alarm sthen,sonst
      SPB   save; // wird nie Unterlast angezeit

      L     2;
      U     #MSG_Min; // Unterlast Alarm
      SPB   save;

      L     8; // Sperre Extern/manuell
      U     #EXT_Inhibit;
      SPB   save;

      L     0;

save: T     #iStatus;

END_FUNCTION_BLOCK

FUNCTION_BLOCK "m7b_VirtualSensor2x"
TITLE =Virtuellen Sensor durch verschieben eines Sensors erzeugen (255)
//Erzeugt einen virtuellen Sensor durch verschieben eines Sensorsignal um Impluse
//eines Encoders, dabei wird die Transportrichtung mit vw/rw berücksichtigt und
//der Sensorwert vorw. mit der positiven Flanke, rückwärts mit negativer Flanke
//des Encoders verarbeitet
//
//Verwendung:
//- virtuelle Sensoron über 4-Puls Sensorring in Transporttischen
//
//AUTOR: Stefan Maag, Dipl.-Ing. (FH) Elektrotechnik
//DATUM: 10/2011
//INTERNET: www.maagic7.de
//
//AENDERUNGSVERMERKE:
//--------------------------------------------------------------------------------
//DATUM        NAME       AENDERUNG
//--------------------------------------------------------------------------------
//16.10.2016   S.Maag     fatalen Fehler P##Buffer Berechnung behoben:
//                        Falsche Bereichskennung ausgeblendet. FB funktionierte
//                        nicht mit Instanz-DB Aufruf, nur über Multiinstanz.
//
//                        Bereichskennung muss aus rel. Adresse aus AR2
//                        entfernt werden, da diese 84 DB ist. Wir benötigen
//                        aber 85 Instanz-DB.
//                        FB gestestet mit direktem Instanz-DB und Multinstanz
//                        2x verschachtelt. Funktion I.O.
//
//16.10.2016   S.Maag     Buffer(15) auf Buffer(7) verkürzt. Da DW (32bit)
//                        verwendet wird, sind 256Byte = 8 Dword nicht 16 DWord
//
//22.08.2016   S.Maag     Fehler P##BUFFER behoben, war ohne Instanzdatenoffset
//                        Varable ptrBUFFER eingeführt.
//                        (!!! Falsche Bereichskennung bei FB Aufruf mit Instanz
//                         DB. Siehe Änderung vom 16.10.2016
//
//16.10.2014   S.Maag     Erweiterung für 2tes Signal
//
//07.10.2014   S.Maag     Buffer von 1xDWORD auf DWORD Array (15) = 255 Bits
//                        erhöht, dadruch Verschiebung von 0..255 statt 0..31
//
//--------------------------------------------------------------------------------
//
//HINWEISE:
AUTHOR : 'S.Maag'
FAMILY : Maagic7
VERSION : 0.1


VAR_INPUT
  SENSOR : BOOL ;	//Sensorsignal
  ENCODER : BOOL ;	//Encodersignal
  vw : BOOL ;	//Richtungssignal Antrieb vw
  rw : BOOL ;	//Richtungssignal Antrieb rs
  IMP_DELAY_1 : INT ;	//Anzahl Impulse der Signalverschiebung
  IMP_DELAY_2 : INT ;	//Anzahl Impulse der Signalverschiebung
END_VAR
VAR_OUTPUT
  SIGNAL1 : BOOL ;	//Sensorsignal um Impuse 1 verschoben
  SIGNAL2 : BOOL ;	//Sensorsignal um Impuse 2 verschoben
END_VAR
VAR
  FP_ENCODER : BOOL ;
  FN_ENCODER : BOOL ;
  ptrBit : DWORD ;
  BUFFER : ARRAY  [0 .. 15 ] OF DWORD ;
END_VAR
VAR_TEMP
  BitToRead : DWORD ;
  IMP_DELAY_CHECKED : DWORD ;
  ptrBUFFER : DWORD ;	//Pointer auf BUFFER korrekt mit Instanzdaten-Offset verrechnet
END_VAR
BEGIN
NETWORK
TITLE =

      SET   ;
      SAVE  ;
      CLR   ;
NETWORK
TITLE =Pointer BUFFER, relativ zu Instanzdaten
//ACHTUNG: indirektes kopieren der Daten von Multiinstanzen über Pointer
//ist nur mit Berücksichtigung des absoluten Instanz-Pointers möglich, da
//die P#-Funktion von Step7 den Pointer nur relativ zu den Daten der aktuellen
//Instanz ermittelt. Dieser relative Pointer muss zum Instanzpointer aus AR2
//addiert werden.
//18.10.2016 S.Maag
//Achtung: Es muss zuerst das Adressregister 2 geladen werden und von dort die
//Bereichskennung ausgeblendet: TAR2 liefert immer Bereichskennung 84 des
//Datenbausteins. P##Buffer liefert 85 "Instanzdatenbaustein als
//Bereichskennung", was direkt die Instanzdaten adressiert.
      TAR2  ; // load Akku with instance pointer
      UD    DW#16#FFFFFF; // Remove highest Byte (memory range / Bereichskennung) = 84 "DB"
      L     P##BUFFER; // load relative address of BUFFER()
      +D    ; // add instance and relative data pointer
      T     #ptrBUFFER; // Pointer Buffer()

NETWORK
TITLE =Signal 1 um IMP_DELAY_1 verschoben aus Puffer lesen

      L     #IMP_DELAY_1; // 00..255 als Delay erlaubt
      L     DW#16#FF; // auf 8 Bit =255 begrenzen
      UD    ;
      T     #IMP_DELAY_CHECKED; // geprüfte Verzögerung max. 8 Bit 0..255

      L     #ptrBit; // akteller Pointer Bit Ringpuffer
      L     #IMP_DELAY_CHECKED; // Auslesedifferenz (Delay)
      -D    ; // BitNoInBuffer - Delay
      L     DW#16#FF; // Limit to 8 Bits (255)
      UD    ;
      T     #BitToRead; // BitNoToRead
      L     #ptrBUFFER; // Adresse Puffer laden
      +D    ; // Bitposition addieren
      LAR1  ; // In Adressregister laden
      U      [AR1,P#0.0]; // in Puffer schreiben
      =     #SIGNAL1; // virtueller Sensor

NETWORK
TITLE =Signal 2 um IMP_DELAY_2 verschoben aus Puffer lesen

      L     #IMP_DELAY_2; // 00..255 als Delay erlaubt
      L     DW#16#FF; // auf 8 Bit =255 begrenzen
      UD    ;
      T     #IMP_DELAY_CHECKED; // geprüfte Verzögerung max. 8 Bit 0..255

      L     #ptrBit; // akteller Pointer Bit Ringpuffer
      L     #IMP_DELAY_CHECKED; // Auslesedifferenz (Delay)
      -D    ; // BitNoInBuffer - Delay
      L     DW#16#FF; // Limit to 8 Bits (255)
      UD    ;
      T     #BitToRead; // BitNoToRead
      L     #ptrBUFFER; // Adresse Puffer laden
      +D    ; // Bitposition addieren
      LAR1  ; // In Adressregister laden
      U      [AR1,P#0.0]; // in Puffer schreiben
      =     #SIGNAL2; // virtueller Sensor

NETWORK
TITLE =Ringpuffer 255 Bit für Sensorsignal

      U     #ENCODER; // Encoder positive Flanke
      FP    #FP_ENCODER;
      U     #vw;
      SPB   p; // vorwärts/positiv

      U     #ENCODER;
      FN    #FN_ENCODER;
      U     #rw; // rückwärts/negativ
      SPB   n;

      BEA   ;

p:    L     #ptrBit; // vorwärts/positiv
      +     L#1; // Pointer Bit +
      SPA   save;

n:    NOP   0; // rückwärts/negativ
      L     #ptrBit; // Pointer Bit -
      +     L#-1;

save: L     DW#16#FF; // max. Bitposition in Puffer (255)
      UD    ; // ptr_Puffer auf max 8Bit (255) begrenzen
      T     #ptrBit; // Pointer aktuelles Bit im Puffer  0..255
      L     #ptrBUFFER; // Adresse Puffer laden
      +D    ; // Bitposition addieren
      LAR1  ; // In Adressregister laden
      U     #SENSOR; // Sensorsingal
      =      [AR1,P#0.0]; // in Ringpuffer schreiben



END_FUNCTION_BLOCK

FUNCTION_BLOCK "m7b_VirtualSensor_32"
TITLE =Erweiterte virtelle Sensorfunktion mit belgter & freier Strecke
//Erzeugt einen virtuellen Sensor durch verschieben eines Sensorsignal um Impluse
//eines Encoders, dabei wird die Transportrichtung mit vw/rw berücksichtigt und
//der Sensorwert vorw. mit der positiven Flanke, rückwärts mit negativer Flanke
//des Encoders verarbeitet.
//Die maximale Verschiebung beträgt 32 Impulse (= den 32 Bits von dwBuffer)
//
//Verwendung:
//- virtuelle Sensoron über 4-Puls Sensorring in Transporttischen
//
//AUTOR: Stefan Maag, Dipl.-Ing. (FH) Elektrotechnik
//DATUM: 10/2011
//INTERNET: www.maagic7.de
//
//AENDERUNGSVERMERKE:
//--------------------------------------------------------------------------------
//DATUM        NAME       AENDERUNG
//--------------------------------------------------------------------------------
//11.01.2018   S.Maag     NW 5: Weg frei nach Sensor nur, wenn Sensor auch frei.
//                        Bisher wurde weg frei gemeldet, wenn Sensor bereits
//                        wieder belegt war, aber noch keine Encoderflanke
//                        auftrat.
//
//08.07.2015   S.Maag     NW 4: bei Reset, NW überspringen und  belegte/freie
//                        Strecke nue berechnen
//--------------------------------------------------------------------------------
//
//HINWEISE:
AUTHOR : 'S.Maag'
FAMILY : Maagic7
VERSION : 0.1


VAR_INPUT
  RESET : BOOL ;	//RESET Befehl
  SENSOR : BOOL ;	//Sensorsignal
  ENCODER : BOOL ;	//Encodersignal
  vw : BOOL ;	//Richtungssignal Antrieb vw
  rw : BOOL ;	//Richtungssignal Antrieb rs
  IMP_DELAY : INT ;	//Anzahl Impulse der Signalverschiebung
END_VAR
VAR_OUTPUT
  SIGNAL : BOOL ;	//Sensorsignal um Impuse verschoben
  IMP_FREI : INT ;
  IMP_BELEGT : INT ;
END_VAR
VAR
  FP_ENCODER : BOOL ;
  FN_ENCODER : BOOL ;
  dwBUFFER : DWORD ;
END_VAR
VAR_TEMP
  cnt_IMP_Hi : INT ;
  cnt_IMP_Lo : INT ;
END_VAR
BEGIN
NETWORK
TITLE =

      SET   ;
      SAVE  ;
      CLR   ;

NETWORK
TITLE =Reset: Alle Sensorbelegungen löschen : dwBuffer := 0

      UN    #RESET; // kein Reset, dann weiter
      SPB   ne2;
      L     DW#16#0; // RESET ausführen: dwBuffer := 0
      T     #dwBUFFER;
ne2:  NOP   0;
NETWORK
TITLE =um IMP_DELAY verschobenen virtullen Sensor aus BUFFER lesen
//Wenn IMP_DELAY = 0, dann wird aktueller Sensorzustand als Signal ausgegeben
//sonst das verschobene Signal aus dwBuffer gelesen
      L     DW#16#FF; // erlaubter wert 0..255
      L     #IMP_DELAY; // 00..32 als Delay erlaubt
      UD    ;
      L     0; // wenn Versatz =0 dann
      <>I   ; // aktuellen Sensorzustand
      SPB   ok; // als Singal ausgeben
      U     #SENSOR;
      =     #SIGNAL;
      SPA   ne3; // VKE wird mitgenommen

ok:   TAK   ; // Versatz nicht 0, dann Versatz zurück in Akku 1
      L     #dwBUFFER; // Buffer laden
      SRD   ; // um Anzahl Bits IMP_DELAY (Wert in Akku 2) schieben
      U     >0; // letztes geschobenes bit ist im Statusregister A1 und kann mit >0 abgefragt werden
      =     #SIGNAL; // virtueller Sensor
ne3:  NOP   0;
NETWORK
TITLE =Ringpuffer 32 Bit für Sensorsignal
//Ringpuffer des Sensorsignals in dwBuffer
//
//08.07.2015 S.Maag : bei RESET NW überspringen - blegt/frei neu berechnen
      U     #RESET; // Bei Reset, freie und belegte Strecke neu berechnen
      SPB   ne4;

      U     #ENCODER; // Encoder positive Flanke
      FP    #FP_ENCODER;
      U     #vw;
      SPB   p; // vorwärts/positiv

      U     #ENCODER;
      FN    #FN_ENCODER;
      U     #rw; // rückwärts/negativ
      SPB   n;

      BEA   ;

n:    L     #dwBUFFER; // Buffer laden
      SRD   1; // für neus Signal bei rückw.: rechts schieben
      T     #dwBUFFER;
      SPA   ne4;

p:    L     #dwBUFFER; // Buffer laden
      SLD   1; // für neues Signal bei vorw.: links schieben
      L     DW#16#1; // High Signal für Sensor belegt!
      OD    ; // Hi mit ODER in Bit_0 eintragen
      U     #SENSOR; // Wenn Sensor belegt
      SPB   save; // dann weiter mit Hi-Signal eintragen
      TAK   ; // Sensor war nicht belegt: SRD 1 Buffer zurück in Akku 2 (neues Bit bleibt Lo)
save: T     #dwBUFFER; // neuer  Buffer
ne4:  NOP   0;

NETWORK
TITLE =Freie und belegte Impulse (Wegstrecke) nach Sensor
//// Strukturporgramm der Funktion
//
//IF dwBUFFER = DW#16#FFFFFFFF THEN   // alle 32 Bits belegt
//   cnt_IMP_Hi = 32   // Belegte Impulse nach Sensor := 32
//   cnt_IMP_Lo = 0
//ELSE_IF dwBUFFER = 0 // kein Bit in dwBuffer belegt
//   cnt_IMP_Hi = 0
//   cnt_IMP_Lo = 32   // min. 32 Impulse freie Wegstrecke nach Sensor
//ELSE
//  IF dwBUFFER.Bit0 = TRUE THEN
//     // Bit0 Hi => Wegstrecke nach Sensor belegt
//     // belegte Wegstrecke besimmen
//    LOPH   // Hi-Bits zählen
//  ELSE  // dwBUFFER.Bit0 = FALSE
//    // Bit0 LO => Wegstrecke nach Sensor frei
//    // freie Wegstrecke besimmen, wenn Sensor nicht belegt
//    IF NOT Sensor THEN
//       LOPL   // Lo-Bits zählen
//    END_IF
//  END_IF
//END_IF

      L     0;
      T     #cnt_IMP_Hi; // Zähler Hi-Impulse auf 0
      T     #cnt_IMP_Lo; // Zähler Lo-Impulse auf 0

      L     DW#16#FFFFFFFF; // Vergleichswert alle Bits Hi
      L     #dwBUFFER; // nur wenn Buffer <>0 und BUFFER <> FFFF FFFF
      <>D   ; // dann Anzahl freie Stellen bestimmen
      SPB   chkZ; // Wenn Buffer nicht alle Bits belegt, dann Check_Zero
      L     32; // Zähler belegte Impulse = 32
      T     #cnt_IMP_Hi;
      SPA   sav;

chkZ: L     L#0; // Vergleichsert alle Bits Lo
      <>D   ; // BUFFER auf 0 prüfen
      SPB   If; // Wenn Buffer auch nicht 0, dann suche nach freier oder belegter Wegstrecke
      L     32; // Wenn Buffer =0, dann sind alle 32 Stellen frei
      T     #cnt_IMP_Lo; // Zähler freie Impulse = 32
      SPA   sav; // und die freie Wegstrecke ist 32 Impulse => speichern

// If BUFFER.Bit0 = Hi THEN GOTO LOPH 'Hi-zählen' ELSE GOTO LOPL 'Lo-zählen'

If:   TAK   ; // BUFFER in AKKU 1 zurück
      PUSH  ; // PUSH kopiert AKKU 1 nach AKKU 2, somit BUFFER in beiden AKKUS
      SRD   1; // BIT_O von BUFFER in STATUSBIT schieben
      L     L#0; // Bitzähler mit 0 laden
      SPN   LOPH; // If BUFFER.Bit0 <>0, dann Schleife Hi-Werte zählen (belegte IMPULSE)

      U     #SENSOR; // IF Sensor is Hi THEN 'no free distance'
      SPB   sav; // Save the 0 values
      SPA   LOPL; // Else Schleife Lo-Werte zählen (freie IMPULSE)

// END_IF

// Schleife Hi-Bits zählen, belegte Wegstrecke nach Sensor
LOPH: TAK   ; // BUFFER zurück in AKKU_1 ; Bitzähler in Akku_2
      SRD   1; // BUFFER ShiftRight: Bit => STATUS A1
      TAK   ; // Bitzähler wieder in Akku 1 (beim ersten Mal 0)
      INC   1; // Bitzähler um 1 erhöhen
      SPZ   savH; // Wenn Bit=0 dann Hi-zählen ENDE: Bitzähler Hi speichern
      SPA   LOPH;
savH: T     #cnt_IMP_Hi; // Bitzähler in Hi-Impulse speichern
      SPA   sav;

// Schleife Lo-Bits zählen, freie Wegstrecke nach Sensor
LOPL: TAK   ; // BUFFER zurück in AKKU_1 ; Bitzähler in Akku_2
      SRD   1; // BUFFER ShiftRight: Bit => STATUS A1
      TAK   ; // Bitzähler wieder in Akku 1 (beim ersten Mal 0)
      INC   1; // Bitzähler um 1 erhöhen
      SPN   savL; // Wenn Bit=1 dann Lo-zählen ENDE: Bitzähler Lo speichern
      SPA   LOPL;
savL: T     #cnt_IMP_Lo; // Bitzähler in Lo-Impulse speichern

sav:  L     #cnt_IMP_Hi; // Zähler Hi-Impulse auf
      T     #IMP_BELEGT; // Ausgang Impulse belegte Wegstrecke

      L     #cnt_IMP_Lo; // Zähler Hi-Impulse auf
      T     #IMP_FREI; // Ausgang Impulse freie Wegstrecke
END_FUNCTION_BLOCK

FUNCTION_BLOCK "m7b_RampTime_INT!!!"
TITLE =Rampe Up/Down über Zeit für INT-Werte
//
//AUTOR: Stefan Maag, Dipl.-Ing. (FH) Elektrotechnik
//DATUM: 4/2009
//INTERNET: www.maagic7.de
//
//AENDERUNGSVERMERKE:
//--------------------------------------------------------------------------------
//DATUM        NAME       AENDERUNG
//--------------------------------------------------------------------------------
//
//--------------------------------------------------------------------------------
//
//HINWEISE:
AUTHOR : 'S.Maag'
FAMILY : Maagic7
VERSION : 0.1


VAR_INPUT
  iSOLL : INT ;	//Sollwert
  iRampMax : INT ;	//Endwert Rampe (Maximalwert)
  iRampMin : INT ;	//Startwert Rampe (Minimalwert)
  timUP : TIME ;	//Zeit Beschleunigungsrampe
  timDOWN : TIME ;	//Zeit Bremsrampe
END_VAR
VAR_OUTPUT
  iOUT : INT ;	//Ausgang aktueller Rampenwert
  DSP_TimeDiff : TIME ;
END_VAR
VAR
  m_rOUT : REAL ;	//letzter Ausgangswert
  m_SysTime : TIME ;	//Systemzeit beim letzten Aufruf
END_VAR
VAR_TEMP
  TimeDiff : TIME ;
  aktSysTime : TIME ;
  rABS_SollDiff : REAL ;
  rRampRange : REAL ;
  RampUp : BOOL ;
  RampDown : BOOL ;
  rTimeFaktor : REAL ;
  rMaxDiffInCycle : DINT ;
END_VAR
BEGIN
NETWORK
TITLE =



NETWORK
TITLE =Zeitdifferenz zum letzten Bausteinaufruf

      CALL "TIME_TCK" (// aktuelle Systemzeit in ms
           RET_VAL                  := #aktSysTime);

      L     #aktSysTime; // aktuelle Systemzeit
      L     #m_SysTime; // Systemzeit beim letzten Aufruf
      UC    "m7b_ABS_DIFF_S7SysTime"; // Absolute Differenz S7-Systemzeiten 31Bit
      T     #TimeDiff; // Absolutwert Zeitdifferenz in ms
      L     L#0; // Wenn keine Zeitdifferenz, dann
      ==D   ; // Baustein ENDE
      BEB   ;
      L     #aktSysTime; // aktuelle Systemzeit
      T     #m_SysTime; // Systemzeit beim letzten Aufruf
      L     #TimeDiff;
      T     #DSP_TimeDiff;


NETWORK
TITLE =Wenn Sollwert & Ausgangswert < iMin, dann keine Rampe
//Out=Soll
      L     #iSOLL;
      L     #iRampMin;
      >I    ;
      SPB   RAMP;
      L     #iOUT;
      L     #iRampMin;
      >I    ;
      SPB   RAMP;

      L     #iSOLL;
      ITD   ;
      DTR   ;
      T     #m_rOUT;
      SPA   END;

RAMP: NOP   0;
NETWORK
TITLE =Beschleunigungs- oder Bermsrampe ?

      L     #iSOLL; // aktueller Sollwert
      L     #iOUT; // letzter Ausgangswert
      >I    ;
      =     #RampUp;
      <I    ;
      =     #RampDown;

NETWORK
TITLE =Rampensteuerbereich ermitteln

      L     #iRampMax;
      L     #iRampMin;
      -I    ;
      ITD   ;
      DTR   ;
      T     #rRampRange;


NETWORK
TITLE =Maximal erlaubte Differenz in diesem Zyklus

      L     #timUP; // Beschleunigungsrampe
      U     #RampUp;
      SPB   calc;
      L     #timDOWN; // oder Bremsrampe
calc: DTR   ;
      L     #TimeDiff;
      DTR   ;
      /R    ;
      T     #rTimeFaktor;

      L     #rRampRange;
      L     #rTimeFaktor;
      /R    ;
      T     #rMaxDiffInCycle;

NETWORK
TITLE =Absolute Differenz von Ausgang und Sollwert

      L     #iOUT;
      L     #iSOLL;
      -I    ;
      SPP   p2;
      NEGI  ;
p2:   ITD   ;
      DTR   ;
      T     #rABS_SollDiff;
NETWORK
TITLE =

      L     #rMaxDiffInCycle;
      L     #rABS_SollDiff;
      >R    ;
      L     #iSOLL;
      ITD   ;
      DTR   ;
      SPB   save;

      U     #RampUp;
      SPB   rup;
      U     #RampDown;
      SPB   rdn;
      SPA   save;

rup:  L     #m_rOUT;
      L     #rMaxDiffInCycle;
      +R    ;
      SPA   save;
rdn:  L     #m_rOUT;
      L     #rMaxDiffInCycle;
      -R    ;
save: T     #m_rOUT;

NETWORK
TITLE =Ausgangswert Ausgeben

END:  L     #iRampMax;
      ITD   ;
      DTR   ;
      L     #m_rOUT; // Real-Wert
      >R    ;
      SPB   sav;
      TAK   ;
      T     #m_rOUT;
sav:  RND   ;
      T     #iOUT; // integer Wert


END_FUNCTION_BLOCK

FUNCTION_BLOCK "m7b_4xMUX_RevSync_INT"
TITLE =4x Schalter-Multiplexer INT, mit Reverse Synchronisierung
//Rückwärts synchronisierender Multiplexer
//
//Mit diesem Baustein lassen sich folgende Probleme beheben, die vor allem bei
//Maschinenumbauten bzw. Erweiterungen auftreten.
//
//- Hinzufügen eines 2ten Bedienpanels, wobei jedoch immer nur ein Panel die
//  Bedienberechtigung hat.
//
//Hiermit lassen sich mehrere Schalter auf einen Schalter synchronisieren. Mit
//cfgSyncSW lassen sich die Schalterstellungen untereinander synchronisieren,
//d.h. der aktive Schalter schaltet die Schalter der anderen Panels mit.
//Ebenfalls lassen sich die Schalter durch den Ausgang rückwärts sychronisieren
//(cfgRevSync). Damit werden die Schalterstellungen dem Ausgangswert nachgeführt.
//Dies ist z.B. notwendig, wenn ein Softwareschalter der z.B. über Multiswitch
//gesteuert wird verwendet wird.
//
//[IN]
//SELECT : Auswahl aktiver Schalter 0: keiner 1: SWITCH_1 2: SWITCH_2 usw.
//cfgSyncSW : Konfiguration Schalter untereinander synchronisieren
//cfgRevSync: Konfiguration Reverse Synchronisation: Schalter mit Ausgang
//            synchronisieren (Ausgang schaltet schalter)
//
//AUTOR: Stefan Maag, Dipl.-Ing. (FH) Elektrotechnik
//DATUM: 7/2011
//INTERNET: www.maagic7.de
//
//AENDERUNGSVERMERKE:
//--------------------------------------------------------------------------------
//DATUM        NAME            AENDERUNG
//--------------------------------------------------------------------------------
//
//--------------------------------------------------------------------------------
//
//HINWEISE: Die Notwendigkeit, die Idee und der erste Umsetzungsversuch stammt
//          bereits von 06/2007
AUTHOR : 'S.Maag'
FAMILY : Maagic7
VERSION : 0.1


VAR_INPUT
  SELECT : INT ;	//Auswahl aktiver Schalter 0: keiner 1: SWITCH_1 2: SWITCH_2 usw.
  cfgSyncSW : BOOL ;	//Konfiguration: Schalter untereinander synchronisieren
  cfgRevSync : BOOL ;	//Konfiguration: Reverse Synchronisation: Schalter mit Ausgang synchronisieren
END_VAR
VAR_IN_OUT
  SWITCH_1 : INT ;
  SWITCH_2 : INT ;
  SWITCH_3 : INT ;
  SWITCH_4 : INT ;
  OUT : INT ;
END_VAR
VAR
  mem_OUT : INT ;
  mem_SWITCH_SEL : INT ;
END_VAR
BEGIN
NETWORK
TITLE =ENO := TRUE

      SET   ;
      SAVE  ;
      CLR   ;
NETWORK
TITLE =Wenn extern veränderter Ausgang, dann RevSync
//Wenn der Ausgnang (OUT) extern verändert wurde, dann die Schalter nachführen,
//sofern ReversSychronisation (RevSync) aktiv.
      UN    #cfgRevSync; // Wenn RevSync nicht aktiv, dann
      SPB   ne2; // überspringen

      L     #mem_OUT; // pruefen, ob Ausgang
      L     #OUT; // extern verändert wurde
      ==I   ; // wenn NEIN, dann weiter
      SPB   ne2;
// Ausgang wurde extern verändert
      T     #mem_OUT; // aktuellen OUT in mem_OUT speichern
      U     #cfgSyncSW; // Wenn Schalter syncronisieren, dann
      SPB   RSAL; // alle auf Ausgang syncronisieren
      SPA   RSY1; // sonst nur aktuellen Schalter syncronisieren

ne2:  NOP   0;

NETWORK
TITLE =RevSync, wenn SWITCH_SEL Multiplexer umgeschaltet wird
//Beim Umschalten des Multiplexers auf einen anderen Eingang, wird zuerst
//Rücksyncronisiert, damit durch das Umschalten keine ungewollten
//Schalthandlungen auftreten.
      L     #mem_SWITCH_SEL; // SWITCH_SEL
      L     #SELECT; // verändert (Multiplexerumschaltung)?
      ==I   ;
      SPB   ne3; // wenn nein, dann weiter
      T     #mem_SWITCH_SEL; // sonst SWITCH_SEL Wert in mem speichern

      UN    #cfgRevSync; // Wenn ReverseSyc aus,
      SPB   ne3; // dann weiter

      U     #cfgSyncSW; // sonst wenn auch Schalter sync.
      SPB   RSAL; // dann alle Schalter auf Ausgang syncronisieren
      SPA   RSY1; // sonst nur aktiven Schalter auf Ausgang sync.

ne3:  NOP   0;

NETWORK
TITLE =4x Multiplexer

      L     #SELECT;
      SPL   SW0;
      SPA   SW0;
      SPA   SW1;
      SPA   SW2;
      SPA   SW3;
      SPA   SW4;

SW0:  BEA   ; // kein Schalter aktiviert

SW1:  L     #SWITCH_1;
      UN    #cfgSyncSW; // Wenn Schalter syncronisieren nicht activ,
      SPB   save; // dann speichern
      T     #SWITCH_2; // sonst restliche Schalter syncronisieren
      T     #SWITCH_3;
      T     #SWITCH_4;
      SPA   save;

SW2:  L     #SWITCH_2;
      UN    #cfgSyncSW;
      SPB   save;
      T     #SWITCH_1;
      T     #SWITCH_3;
      T     #SWITCH_4;
      SPA   save;

SW3:  L     #SWITCH_3;
      UN    #cfgSyncSW;
      SPB   save;
      T     #SWITCH_1;
      T     #SWITCH_2;
      T     #SWITCH_4;
      SPA   save;

SW4:  L     #SWITCH_4;
      UN    #cfgSyncSW;
      SPB   save;
      T     #SWITCH_1;
      T     #SWITCH_2;
      T     #SWITCH_3;

save: T     #OUT;
      T     #mem_OUT;
      BEA   ;
NETWORK
TITLE =Reverse Sync - nur aktiven Schalter
//aktiven Schalter rücksyncronisieren (Schaltereingang = aktueller OUT)
RSY1: L     #SELECT;
      SPL   RSW0; // Sprungziel bei Overflow: SWITCH_SEL>4
      SPA   RSW0; // 0, kein Eingang ausgewählt
      SPA   RSW1;
      SPA   RSW2;
      SPA   RSW3;
      SPA   RSW4;

RSW0: BEA   ; // kein Schalter aktiviert

RSW1: L     #OUT; // RevSync Switch 1
      T     #SWITCH_1;
      BEA   ;

RSW2: L     #OUT; // RevSync Switch 2
      T     #SWITCH_2;
      BEA   ;

RSW3: L     #OUT; // RevSync Switch 3
      T     #SWITCH_3;
      BEA   ;

RSW4: L     #OUT; // RevSync Switch 4
      T     #SWITCH_4;
      BEA   ;
NETWORK
TITLE =Reverse Sync - alle Schalter

RSAL: L     #OUT;
      T     #SWITCH_1;
      T     #SWITCH_2;
      T     #SWITCH_3;
      T     #SWITCH_4;

END_FUNCTION_BLOCK

FUNCTION_BLOCK "m7b_RAMP_LIN_TIME"
TITLE =Linear-Rampen-Generator über Zeit
//Generiert eine lineare Rampe zwischen den Geschwindigkeiten MIN und MAX.
//
//AUTOR: Stefan Maag, Dipl.-Ing. (FH) Elektrotechnik
//DATUM: 5/2012
//INTERNET: www.maagic7.de
//
//AENDERUNGSVERMERKE:
//--------------------------------------------------------------------------------
//DATUM        NAME          AENDERUNG
//--------------------------------------------------------------------------------
//03/12/2013   S.Maag      SFC64 TimeTick Zeitdifferenz korrigiert
//                         da 31Bit, Fehler bei Überlauf. Auf 32 Bit-Rechnung
//                         erweitert
//--------------------------------------------------------------------------------
//
//HINWEISE:
AUTHOR : 'S.Maag'
FAMILY : Maagic7
VERSION : 0.1


VAR_INPUT
  RESET : BOOL ;	//Reset Speed to SetPoint
  Speed_SetPoint : INT ;
  Speed_min : INT ;	//Geschwindigkeit minimal
  Speed_max : INT ;	//Geschwindigkeit maximal
  ACC_TIME : TIME ;	//Acceleration Time (min to max)
  DECC_TIME : TIME ;	//Decceleration Time (max to min)
  TIME_BASE : TIME ;
END_VAR
VAR_OUTPUT
  Speed : INT ;
  MSG_ACC : BOOL ;	//Meldung Beschleunigung
  MSG_DECC : BOOL ;	//Meldung Verzögerung
END_VAR
VAR
  r_memSpeed : REAL ;
  memTime : TIME ;
END_VAR
VAR_TEMP
  rACC_STEP : REAL ;
  rDECC_STEP : REAL ;
  rSPEEDDIFFxTIMEBASE : DINT ;
  aktSysTime : TIME ;
  TimeDiff : TIME ;
  rSpeedSetPoint : REAL ;
END_VAR
BEGIN
NETWORK
TITLE =



NETWORK
TITLE =prüfen auf abgelaufene Zeitbasis und Resetverarbeitung

      CALL "TIME_TCK" (
           RET_VAL                  := #aktSysTime);

      UN    #RESET; // Wenn Reset,
      SPB   do;
      R     #MSG_ACC;
      R     #MSG_DECC;
      L     #aktSysTime; // dann
      T     #memTime;
      L     #Speed_SetPoint; // SetPoint als Speed speichern
      SPA   SAVE;

do:   L     #aktSysTime; // aktuelle Systemzeit
      L     #memTime; // gespeicherte Zeit
      UC    "m7b_ABS_DIFF_S7SysTime";
      T     #TimeDiff;
      L     #TIME_BASE; // Zeitbasis
      <D    ; // TimeDiff < TimeBase
      BEB   ; // dann Ende
      L     #aktSysTime;
      T     #memTime; // als letzte Zeit speichern

NETWORK
TITLE =Rampenstufung für beschleunigen & bremsen berechnen
//Beispiel für Berechnung der Beschleunigungsrampe, gleiches gilt für bremsen
//
//STEPS = ACC_TIME/TimeBase  // Anzahl der Rampenstufen
//ACC_STEP = SpeedDiff / (ACC_TIME/TimeBase) = SpeedDiff * TimeBase / ACC_TIME
//
      L     #Speed_max; // Maximalgeschwindigkeit
      L     #Speed_min; // Minimalgeschwindigkeit
      -I    ; // SPEED_DIFF
      ITD   ;
      L     #TIME_BASE;
      *D    ;
      DTR   ;
      T     #rSPEEDDIFFxTIMEBASE;
      L     #ACC_TIME;
      DTR   ;
      /R    ;
      T     #rACC_STEP; // Beschleunigungsstufe


      L     #rSPEEDDIFFxTIMEBASE;
      L     #DECC_TIME;
      DTR   ;
      /R    ;
      T     #rDECC_STEP; // Bremsstufe

NETWORK
TITLE =Beschleunigen oder bremsen?

      L     #Speed_SetPoint; // aktueller Speed Sollwert
      ITD   ;
      DTR   ;
      T     #rSpeedSetPoint; // Real SpeedSetPoint

      L     #Speed_SetPoint;
      L     #r_memSpeed; // Speicher letzter Speed
      RND   ;
      >I    ; // Wenn SetPoint > memSpeed
      SPB   acc; // dann beschleuchnigen
      <I    ; // Wenn SetPoint < memSpeed
      SPB   decc; // dann bremsen
      R     #MSG_ACC;
      R     #MSG_DECC;
      L     #rSpeedSetPoint; // aktueller Speed Sollwert
      SPA   SAVE;

acc:  S     #MSG_ACC;
      R     #MSG_DECC;
      L     #r_memSpeed; // Beschleunigen
      L     #rACC_STEP; // um eine Stufe
      +R    ;
      L     #rSpeedSetPoint; // bei Beschleunigung
      >R    ; // auf max SetPoint
      SPB   SAVE; // begrenzen
      TAK   ;
      SPA   SAVE;

decc: S     #MSG_DECC;
      R     #MSG_ACC;
      L     #r_memSpeed; // Bremsen
      L     #rDECC_STEP; // um eine Stufe
      -R    ;
      L     #rSpeedSetPoint; // bei Verzögerung
      <R    ; // auf min SetPoint
      SPB   SAVE; // begrenzen
      TAK   ;
      SPA   SAVE;

NETWORK
TITLE =nun noch auf Maximalwert begrenzen

SAVE: L     #Speed_max; // Speed max
      ITD   ;
      DTR   ;
      >R    ; // Wenn SpeedAkt >  MaxSpeed,
      SPB   sav; // dann MaxSpeed speichern
      TAK   ; // sonst SpeedAkt zurück in Akku1
      L     #Speed_min; // Wenn SpeedAct < MinSpeed,
      ITD   ;
      DTR   ;
      <R    ; // dann MinSpeed speichern
      SPB   sav;
      TAK   ; // sonst SpeedAkt zurück in Akku1
sav:  T     #r_memSpeed;
      RND   ;
      T     #Speed; // Speed speichern
      SAVE  ;
END_FUNCTION_BLOCK

FUNCTION_BLOCK "m7b_1of4DeviceEnable"
TITLE =1of4_DeviceEnable
//Enables 1 of 4 devices.
//Allows only 1 device to be enabled.
//Changes the device enable with adjustable delay
//
//AUTOR: Stefan Maag, Dipl.-Ing. (FH) Elektrotechnik
//DATUM: 08/2013
//INTERNET: www.maagic7.de
//
//AENDERUNGSVERMERKE:
//--------------------------------------------------------------------------------
//DATUM        NAME            AENDERUNG
//--------------------------------------------------------------------------------
//
//--------------------------------------------------------------------------------
//
//HINWEISE: Entwickelt für Schieber Bioabfallaufbereitung
AUTHOR : 'S.Maag'
FAMILY : Maagic7
VERSION : 0.1


VAR_INPUT
  REQ1 : BOOL ;	//Request for Device 1
  REQ2 : BOOL ;	//Request for Device 2
  REQ3 : BOOL ;	//Request for Device 3
  REQ4 : BOOL ;	//Request for Device 3
  timDelay : TIME ;
END_VAR
VAR_OUTPUT
  EN1 : BOOL ;
  EN2 : BOOL ;
  EN3 : BOOL ;
  EN4 : BOOL ;
END_VAR
VAR
  Q_TOF_ENABLE : BOOL ;
  TOF_ENABLE : "TOF";
END_VAR
VAR_TEMP
  tmpEnIsOn : BOOL ;
END_VAR
BEGIN
NETWORK
TITLE =




NETWORK
TITLE =DELAYED ENABLE OFF
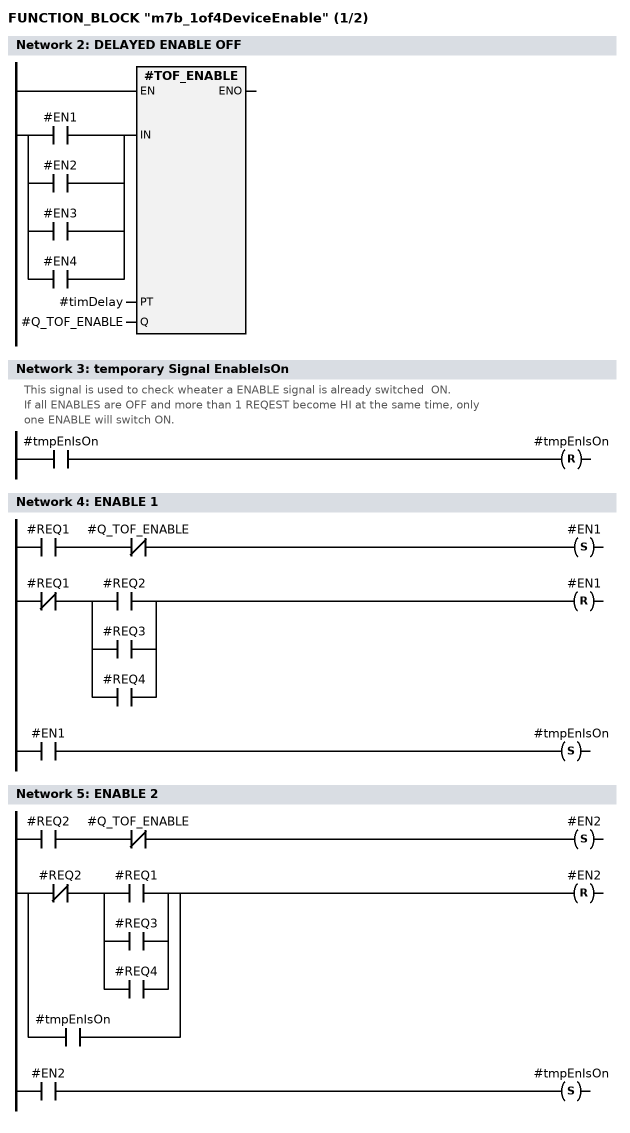



      U(    ;
      O     #EN1;
      O     #EN2;
      O     #EN3;
      O     #EN4;
      )     ;
      =     L      1.0;
      BLD   103;
      CALL #TOF_ENABLE (
           IN                       := L      1.0,
           PT                       := #timDelay,
           Q                        := #Q_TOF_ENABLE);

      NOP   0;
NETWORK
TITLE =temporary Signal EnableIsOn
//This signal is used to check wheater a ENABLE signal is already switched  ON.
//If all ENABLES are OFF and more than 1 REQEST become HI at the same time, only
//one ENABLE will switch ON.
      U     #tmpEnIsOn;
      R     #tmpEnIsOn;
NETWORK
TITLE =ENABLE 1

      U     #REQ1;
      UN    #Q_TOF_ENABLE;
      S     #EN1;
      UN    #REQ1;
      U(    ;
      O     #REQ2;
      O     #REQ3;
      O     #REQ4;
      )     ;
      R     #EN1;
      U     #EN1;
      S     #tmpEnIsOn;
NETWORK
TITLE =ENABLE 2

      U     #REQ2;
      UN    #Q_TOF_ENABLE;
      S     #EN2;
      U(    ;
      UN    #REQ2;
      U(    ;
      O     #REQ1;
      O     #REQ3;
      O     #REQ4;
      )     ;
      O     #tmpEnIsOn;
      )     ;
      R     #EN2;
      U     #EN2;
      S     #tmpEnIsOn;
NETWORK
TITLE =ENABLE 3
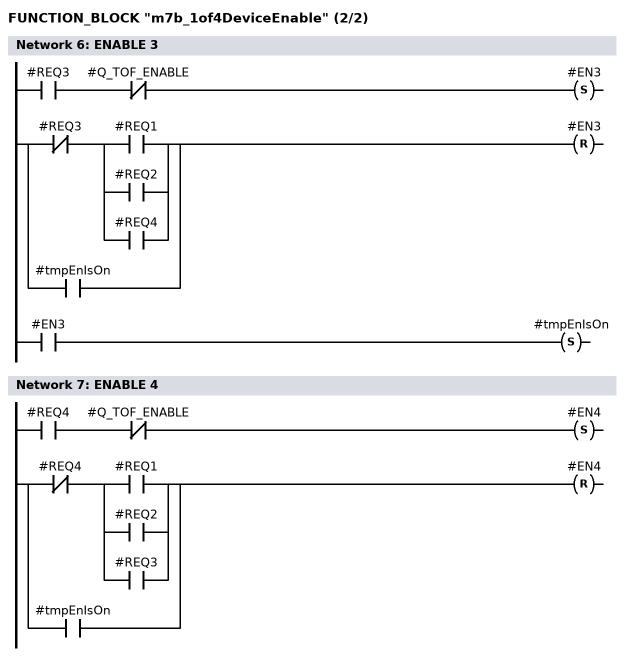

      U     #REQ3;
      UN    #Q_TOF_ENABLE;
      S     #EN3;
      U(    ;
      UN    #REQ3;
      U(    ;
      O     #REQ1;
      O     #REQ2;
      O     #REQ4;
      )     ;
      O     #tmpEnIsOn;
      )     ;
      R     #EN3;
      U     #EN3;
      S     #tmpEnIsOn;
NETWORK
TITLE =ENABLE 4

      U     #REQ4;
      UN    #Q_TOF_ENABLE;
      S     #EN4;
      U(    ;
      UN    #REQ4;
      U(    ;
      O     #REQ1;
      O     #REQ2;
      O     #REQ3;
      )     ;
      O     #tmpEnIsOn;
      )     ;
      R     #EN4;
      NOP   0;
END_FUNCTION_BLOCK

FUNCTION_BLOCK "m7b_PumpPressureMonitor"
TITLE =Pressure monitoring for pumps / Drucküberwachung Pumpen
//Überwachung auf Unterdruck (Trockenlauf/Wassermangel bzw. Rohrbruch)
//Überwachung auf Überdruck (z.B. geschlossene Schieber)
//
//AUTOR: Stefan Maag, Dipl.-Ing. (FH) Elektrotechnik
//DATUM: 08/2012
//
//AENDERUNGSVERMERKE:
//--------------------------------------------------------------------------------
//DATUM        NAME       AENDERUNG
//--------------------------------------------------------------------------------
//04.08.2018   S.Maag    Dokumentation ergänzt/überarbeitet
//
//15.04.2016   S.Maag    SET SAVE CLR in letzte NW verschoben, da ENO nicht TRUE
//                       war. (wird wahrscheinlich von TON-Aufrufen überschrieben)
AUTHOR : 'S.Maag'
FAMILY : Maagic7
VERSION : 0.1


VAR_INPUT
  MSG_RUN : BOOL ;	//Message Pump run
  RESET : BOOL ;	//Error Reset
  rPact : REAL ;	//actual pressure
  rPmin : REAL ;	//minimal pressure
  rPmax : REAL ;	//maximal pressure
  timPmin : TIME  := T#30S;	//Time for min pressure Error
  timPmax : TIME  := T#5MS;	//Time for max pressure Error
END_VAR
VAR_OUTPUT
  MSG_ERR : BOOL ;	//ERROR / FAULT (Lo or Hi)
  MSG_ERR_Lo : BOOL ;	//Low pressure error
  MSG_ERR_Hi : BOOL ;	//Over pressure error
  rP_ERR : REAL ;	//Pressure value when error occurs
END_VAR
VAR
  FP_ERR_Pmin : BOOL ;	//Rising edge of low pressure error
  FP_ERR_Pmax : BOOL ;	//Rising edge of over pressure error
  TON_Pmin : "TON";	//Delay low pressure error
  TON_Pmax : "TON";	//Delay over pressure error
END_VAR
VAR_TEMP
  Q_TON_Pmin : BOOL ;
  Q_TON_Pmax : BOOL ;
  DSP_TPmin : TIME ;
  DSP_TPmax : TIME ;
END_VAR
BEGIN
NETWORK
TITLE =Low pressure / Unterdruck
//======================================================================
//              L O W   P R E S S U R E  /  U N T E R D R U C K
//======================================================================
NETWORK
TITLE =Lo pressure check / Auf Unterdruck prüfen (verzögert)



      U     #MSG_RUN;
      U(    ;
      L     #rPact;
      L     #rPmin;
      <R    ;
      )     ;
      UN    #MSG_ERR_Lo;
      =     L     10.0;
      BLD   103;
      CALL #TON_Pmin (
           IN                       := L     10.0,
           PT                       := #timPmin,
           Q                        := #Q_TON_Pmin,
           ET                       := #DSP_TPmin);
      NOP   0;
NETWORK
TITLE =Low pressure Error / Unterdruckstörung

      U(    ;
      U     #Q_TON_Pmin;
      S     #MSG_ERR_Lo;
      U     #RESET;
      R     #MSG_ERR_Lo;
      U     #MSG_ERR_Lo;
      )     ;
      FP    #FP_ERR_Pmin;
      SPBNB _001;
      L     #rPact;
      T     #rP_ERR;
_001: NOP   0;
NETWORK
TITLE =Over pressure / Überdruck
//======================================================================
//          O V E R   P R E S S U R E   /   Ü B E R D R U C K
//======================================================================
NETWORK
TITLE =Over pressure check / Auf Überdruck prüfen (verzögert)

      U     #MSG_RUN;
      U(    ;
      L     #rPact;
      L     #rPmax;
      >R    ;
      )     ;
      UN    #MSG_ERR_Hi;
      =     L     10.0;
      BLD   103;
      CALL #TON_Pmax (
           IN                       := L     10.0,
           PT                       := #timPmax,
           Q                        := #Q_TON_Pmax,
           ET                       := #DSP_TPmax);
      NOP   0;
NETWORK
TITLE =Over pressure Error / Überdruckstörung

      U(    ;
      U     #Q_TON_Pmax;
      S     #MSG_ERR_Hi;
      U     #RESET;
      R     #MSG_ERR_Hi;
      U     #MSG_ERR_Hi;
      )     ;
      FP    #FP_ERR_Pmax;
      SPBNB _002;
      L     #rPact;
      T     #rP_ERR;
_002: NOP   0;
NETWORK
TITLE =ERROR output / Ausgang Störung

      O     #MSG_ERR_Lo;
      O     #MSG_ERR_Hi;
      =     #MSG_ERR;
NETWORK
TITLE =

      SET   ;
      SAVE  ;
      CLR   ;

END_FUNCTION_BLOCK

FUNCTION_BLOCK "m7b_PumpTempMonitor"
TITLE =Temperature monitoring for pumps / Temperaturüberwachung Pumpen
//Stator Temperatur monitoring for pumps with Stator-Temperatur-Sensor
//
//AUTOR: Stefan Maag, Dipl.-Ing. (FH) Elektrotechnik
//DATUM: 03/2019
//
//AENDERUNGSVERMERKE:
//--------------------------------------------------------------------------------
//DATUM        NAME       AENDERUNG
//--------------------------------------------------------------------------------
//
AUTHOR : 'S.Maag'
FAMILY : Maagic7
VERSION : 0.1


VAR_INPUT
  MSG_RUN : BOOL ;	//Message Pump run
  RESET : BOOL ;	//Error Reset
  rStatorTemp : REAL ;	//actual Stator Temperature
  rMediumTemp : REAL ;	//actual Medium Temperature
  rTempOffset : REAL ;	//Allowed Temperature Offset (TempStator > TempMedium)
  timTempMax : TIME  := T#5MS;	//Time for max Temperautre Error
END_VAR
VAR_OUTPUT
  MSG_ERR : BOOL ;	//ERROR / FAULT
  rTemp_ERR : REAL ;	//Stator Temperature value when error occurs
END_VAR
VAR
  m_TempMax : REAL ;
  TON_TempMax : "TON";	//Delay over pressure error
  FP_ERR : BOOL ;	//Rising edge of over pressure error
END_VAR
VAR_TEMP
  Q_TON_TempMax : BOOL ;
  DSP_TempMax : TIME ;
END_VAR
BEGIN
NETWORK
TITLE =

NETWORK
TITLE =Calculate max. allowed Stator Temp. = MediumTemp + Offset
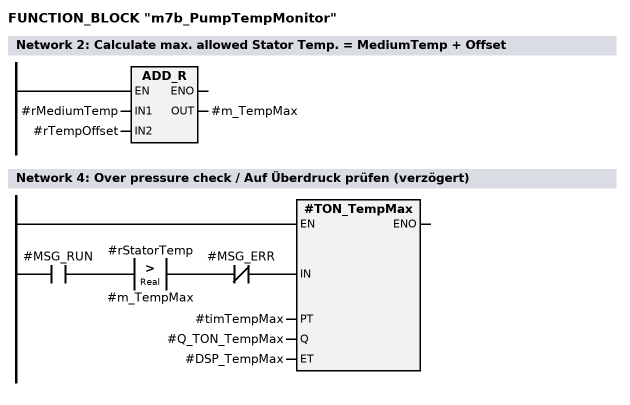

      L     #rMediumTemp;
      L     #rTempOffset;
      +R    ;
      T     #m_TempMax;
      NOP   0;
NETWORK
TITLE =Over Temperature/ Übertemperatur
//======================================================================
//  O V E R   T E M P E R A T U R E   /   Ü B E R T E M P E R A T U R
//======================================================================
NETWORK
TITLE =Over pressure check / Auf Überdruck prüfen (verzögert)

      U     #MSG_RUN;
      U(    ;
      L     #rStatorTemp;
      L     #m_TempMax;
      >R    ;
      )     ;
      UN    #MSG_ERR;
      =     L      6.0;
      BLD   103;
      CALL #TON_TempMax (
           IN                       := L      6.0,
           PT                       := #timTempMax,
           Q                        := #Q_TON_TempMax,
           ET                       := #DSP_TempMax);
      NOP   0;
NETWORK
TITLE =Over temperature Error / Störung Übertemperatur

      U(    ;
      U     #Q_TON_TempMax;
      S     #MSG_ERR;
      U     #RESET;
      R     #MSG_ERR;
      U     #MSG_ERR;
      )     ;
      FP    #FP_ERR;
      SPBNB _001;
      L     #rStatorTemp;
      T     #rTemp_ERR;
_001: NOP   0;
NETWORK
TITLE =

      SET   ;
      SAVE  ;
      CLR   ;

END_FUNCTION_BLOCK

FUNCTION_BLOCK "m7b_DriveError_AutoReset"
TITLE =DriveError AUTO-RESET
//AutoReset the Drives Frequency converter a few times.
//
//[IN]
//MSG_DRIVE_ERR : indicates Drive Fault
//ERR_RESET     : External button to RESET Errors, must be pressed by Operator
//MaxNoOfResets : Max no of Resets allowed during monitoring time (typical 3)
//timResetMonitoring : Time for RESET Monitoring:
//                     during this time only MaxNoOfResets are allowed
//timResetDelay  : Dealy between MsgDriveErr and FC_RESET_Impuls
//timResetImpuls : Duration of FC_RESET_Impuls
//
//[OUT]
//FC_RESET_IMP  : Impuls with duration timResetImpuls to reset frequncy converter
//evt_RESET     : 1 Cycle Event signal: can be used to save time stamp of RESET
//ERR_RESET_CNT : Shows the Error-Reset Counter
//DSP_MonitoringTime : Shows the elappsed time since first RESET
//                    (=ResetMonitoringTime)
//
//
//AUTOR: Stefan Maag, Dipl.-Ing. (FH) Elektrotechnik
//DATUM: 03/2019
//
//AENDERUNGSVERMERKE:
//--------------------------------------------------------------------------------
//DATUM        NAME       AENDERUNG
//--------------------------------------------------------------------------------
//
AUTHOR : 'S.Maag'
FAMILY : Maagic7
VERSION : 0.1


VAR_INPUT
  MSG_DRIVE_ERR : BOOL ;	//Message Drive Error
  ERR_RESET : BOOL ;
  MaxNoOfResets : INT ;	//Maximal number of RESETs during monitoring time
  timResetMonitoring : TIME ;	//Duration of Reset Monitoring
  timResetDelay : TIME ;	//Delay for Reset Impuls, after Error occured
  timResetImpuls : TIME  := T#500MS;	//Duration of Reset Impuls
END_VAR
VAR_OUTPUT
  FC_RESET_IMP : BOOL ;	//Frequency converter RESET Impuls
  evt_RESET : BOOL ;	//Reset Event: can be used to save TimeStamp of Reset
  ERR_RESET_CNT : INT ;	//Counter of Resets
  DSP_MonitoringTime : TIME ;	//Elappsed time since first RESET (Reset monitoring time)
END_VAR
VAR
  TON_RESET_DELAY : "TON";
  TP_RESET : "TP";
  TON_ResetTimeRange : "TP";
  CTU_ERR : "CTU";
  Q_TON_RESET_DELAY : BOOL ;
  Q_TP_RESET : BOOL ;
  Q_TON_ResetTimeRange : BOOL ;
  Q_CTU_Errors : BOOL ;
  m_StartTimeRange : BOOL ;
  m_MaxNoOfResetReached : BOOL ;
  cmd_RESET : BOOL ;	//Reset command for Monitoring Time & RESET-Counter
END_VAR
VAR_TEMP
  DSP_ResetTimeRange : TIME ;
END_VAR
BEGIN
NETWORK
TITLE =

NETWORK
TITLE =Delay Time for Reset when Error occured

      U     #MSG_DRIVE_ERR;
      =     L      4.0;
      BLD   103;
      CALL #TON_RESET_DELAY (
           IN                       := L      4.0,
           PT                       := #timResetDelay,
           Q                        := #Q_TON_RESET_DELAY);

      NOP   0;
NETWORK
TITLE =Create the Output RESET-Impuls for the Frequency converter

      U(    ;
      U     #Q_TON_RESET_DELAY;
      =     L      4.0;
      BLD   103;
      CALL #TP_RESET (
           IN                       := L      4.0,
           PT                       := #timResetImpuls,
           Q                        := #Q_TP_RESET);

      U     BIE;
      )     ;
      U     #Q_TP_RESET;
      =     #FC_RESET_IMP;
NETWORK
TITLE =Start ResetTimeRange Monitoring
//Überwachungszeit für Max. Anzahl der Resets starten.
//
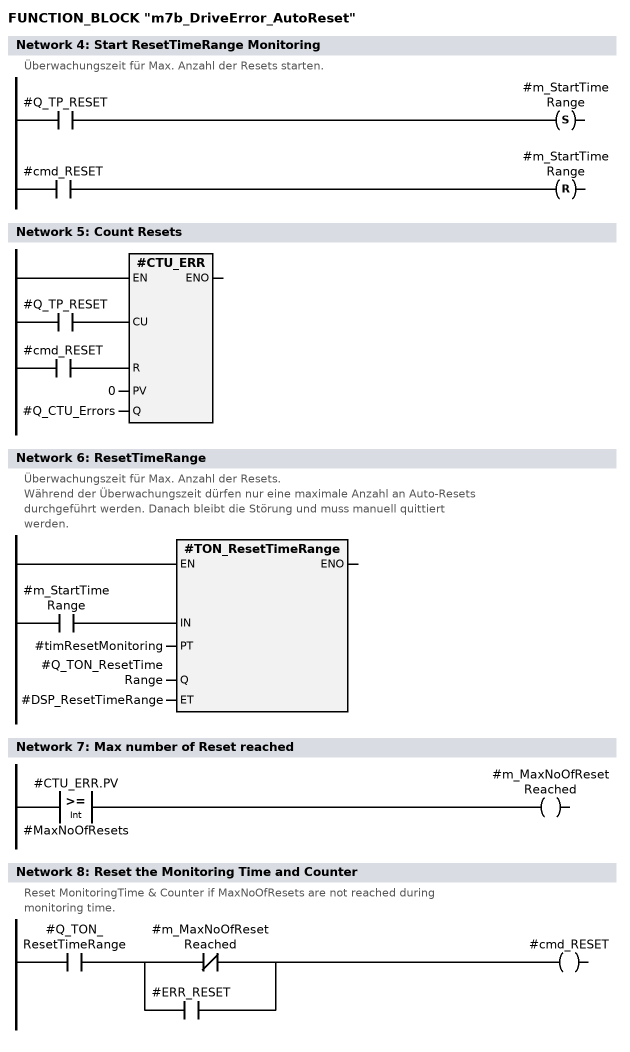
      U     #Q_TP_RESET;
      S     #m_StartTimeRange;
      U     #cmd_RESET;
      R     #m_StartTimeRange;
      NOP   0;
NETWORK
TITLE =Count Resets

      U     #Q_TP_RESET;
      =     L      4.0;
      BLD   103;
      U     #cmd_RESET;
      =     L      4.1;
      BLD   103;
      CALL #CTU_ERR (
           CU                       := L      4.0,
           R                        := L      4.1,
           PV                       := 0,
           Q                        := #Q_CTU_Errors);

      NOP   0;
NETWORK
TITLE =ResetTimeRange
//Überwachungszeit für Max. Anzahl der Resets.
//Während der Überwachungszeit dürfen nur eine maximale Anzahl an Auto-Resets
//durchgeführt werden. Danach bleibt die Störung und muss manuell quittiert
//werden.
      U     #m_StartTimeRange;
      =     L      4.0;
      BLD   103;
      CALL #TON_ResetTimeRange (
           IN                       := L      4.0,
           PT                       := #timResetMonitoring,
           Q                        := #Q_TON_ResetTimeRange,
           ET                       := #DSP_ResetTimeRange);
      NOP   0;
NETWORK
TITLE =Max number of Reset reached

      L     #CTU_ERR.PV;
      L     #MaxNoOfResets;
      >=I   ;
      =     #m_MaxNoOfResetReached;
NETWORK
TITLE =Reset the Monitoring Time and Counter
//Reset MonitoringTime & Counter if MaxNoOfResets are not reached during
//monitoring time.
      U     #Q_TON_ResetTimeRange;
      U(    ;
      ON    #m_MaxNoOfResetReached;
      O     #ERR_RESET;
      )     ;
      =     #cmd_RESET;
END_FUNCTION_BLOCK

FUNCTION_BLOCK "m7b_DriveRuntimeMonitor"
TITLE =Runtime Monitoring Drives / Laufzeitüberwachung Antriebe
//Runtime monitoring of Drives with seperate monitoring time for
//Auto and Manual mode.
//
//In Manual Mode, the STOP command is activated when MaxTime is elapsed.
//In Auto Mode, the STOP command is activated and an ERROR is set. This
//Error must be reset by operator.
//
//AUTOR: Stefan Maag, Dipl.-Ing. (FH) Elektrotechnik
//DATUM: 03/2019
//
//AENDERUNGSVERMERKE:
//--------------------------------------------------------------------------------
//DATUM        NAME       AENDERUNG
//--------------------------------------------------------------------------------
//
AUTHOR : 'S.Maag'
FAMILY : Maagic7
VERSION : 0.1


VAR_INPUT
  MSG_RUN : BOOL ;
  MSG_AUTO : BOOL ;
  RESET : BOOL ;
  timMax_HAND : TIME ;
  timMax_AUTO : TIME ;
END_VAR
VAR_OUTPUT
  CMD_STOP : BOOL ;
  MSG_ERR : BOOL ;
  timRUN : TIME ;
  timREST : TIME ;
END_VAR
VAR
  m_timMaxRun : TIME ;
  TON_MAX_RUN : "TON";
  Q_TON_MAX_RUN : BOOL ;
  m_ERROR : BOOL ;
END_VAR
VAR_TEMP
  xVOID : BOOL ;
  DSP_TON_MAX_RUN : TIME ;
END_VAR
BEGIN
NETWORK
TITLE =

NETWORK
TITLE =Multiplexer for Maximum Runtime in AUTO & HAND

      O(    ;
      UN    #MSG_AUTO;
      SPBNB _001;
      L     #timMax_HAND;
      T     #m_timMaxRun;
      SET   ;
      SAVE  ;
      CLR   ;
_001: U     BIE;
      )     ;
      O(    ;
      U     #MSG_AUTO;
      SPBNB _002;
      L     #timMax_AUTO;
      T     #m_timMaxRun;
      SET   ;
      SAVE  ;
      CLR   ;
_002: U     BIE;
      )     ;
      =     #xVOID;
NETWORK
TITLE =Timer Max Runtime

      U(    ;
      U     #MSG_RUN;
      =     L      6.0;
      BLD   103;
      CALL #TON_MAX_RUN (
           IN                       := L      6.0,
           PT                       := #m_timMaxRun,
           Q                        := #Q_TON_MAX_RUN,
           ET                       := #DSP_TON_MAX_RUN);
      U     BIE;
      )     ;
      U     #Q_TON_MAX_RUN;
      =     #CMD_STOP;
NETWORK
TITLE =FC-Output: timRUN & timREST
//Display at FC-Output:
//- the actual running time (timRUN)
//- the remaining time to Stop (and Error in Auto-Mode)
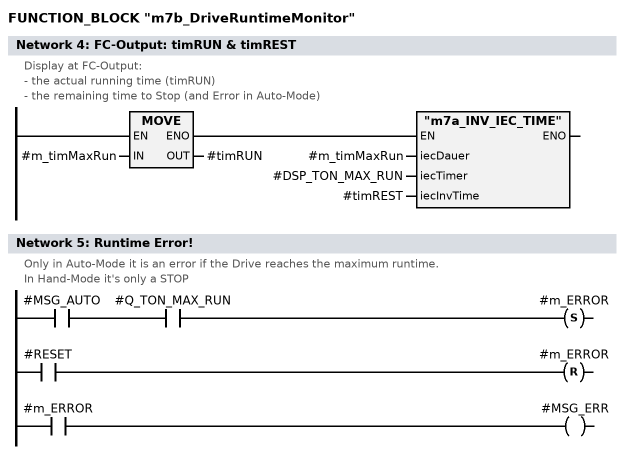
      U(    ;
      L     #m_timMaxRun;
      T     #timRUN;
      SET   ;
      SAVE  ;
      CLR   ;
      U     BIE;
      )     ;
      SPBNB _003;
      CALL "m7a_INV_IEC_TIME" (
           iecDauer                 := #m_timMaxRun,
           iecTimer                 := #DSP_TON_MAX_RUN,
           iecInvTime               := #timREST);
_003: NOP   0;
NETWORK
TITLE =Runtime Error!
//Only in Auto-Mode it is an error if the Drive reaches the maximum runtime.
//In Hand-Mode it's only a STOP
      U     #MSG_AUTO;
      U     #Q_TON_MAX_RUN;
      S     #m_ERROR;
      U     #RESET;
      R     #m_ERROR;
      U     #m_ERROR;
      =     #MSG_ERR;
END_FUNCTION_BLOCK

FUNCTION_BLOCK "m7b_AVERAGE"
TITLE =Mittelwertbildung: 1,3,5,15 Minuten
//Mittelwertbildung von analogen Signalen.
//Verwendung bei Energieerfassung z.B. Strom-, Gas-, Wärmemengenzähler
//
//TAKT_1S: S7 Systemtaktmerker 1-Sekunde
//RESET :  RESET
//rVALUE : Eingangswert
//
//ENO: TRUE
//
//AUTOR: Stefan Maag, Dipl.-Ing. (FH) Elektrotechnik
//DATUM: 11/2013
//INTERNET: www.maagic7.de
//
//AENDERUNGSVERMERKE:
//--------------------------------------------------------------------------------
//DATUM        NAME        AENDERUNG
//--------------------------------------------------------------------------------
//16.10.2016   S.Maag     fatalen Fehler P##Buffer Berechnung behoben:
//                        Falsche Bereichskennung ausgeblendet. FB funktionierte
//                        nicht mit Instanz-DB Aufruf, nur über Multiinstanz.
//
//                        Bereichskennung muss aus rel. Adresse aus AR2
//                        entfernt werden, da diese 84 DB ist. Wir benötigen
//                        aber 85 Instanz-DB.
//                        Code getestet mit FB1141: direkter Instanz-DB und
//                        Multinstanz mit 2x Verschachtelung. Funktion I.O.
//--------------------------------------------------------------------------------
//
//HINWEISE:
AUTHOR : 'S.Maag'
FAMILY : Maagic7
VERSION : 0.1


VAR_INPUT
  TAKT_1S : BOOL ;	//Taktgeber: (Flankenauswertung erfolgt im FB)
  RESET : BOOL ;	//RESET: Zähler rücksetzen
  rVALUE : REAL ;	//Zu integrierender WERT
END_VAR
VAR_OUTPUT
  rAVG_1min : REAL ;	//1 Minuten Mittelwert
  rAVG_3min : REAL ;	//3 Minuten Mittelwert
  rAVG_5min : REAL ;	//5 Minuten Mittelwert
  rAVG_15min : REAL ;	//15 Minuten Mittelwert
  evtNewValues : BOOL ;	//Ereignis Werte aktualisiert
  DSP_BUFFER_INDEX : INT ;	//Anzeige Buffer Index ARRAY[INDEX]
END_VAR
VAR
  HM_FP_TAKT : BOOL ;	//Lokaler Speicher:
  CNT_SEC : INT ;
  CNT_MIN : INT ;
  dIDX : DINT ;
  memSum1min : REAL ;	//Integralwert
  rARRAY : ARRAY  [0 .. 15 ] OF REAL ;
END_VAR
VAR_TEMP
  tmp_rAVG : REAL ;
  ptrARRAY : DWORD ;
  I : INT ;
  dJ : DINT ;
  tmp_rSUM : REAL ;
END_VAR
BEGIN
NETWORK
TITLE =Absoluten Pointer auf ARRAY berechnen
//18.10.2016 S.Maag
//Achtung: Es muss zuerst das Adressregister 2 geladen werden und von dort die
//Bereichskennung ausgeblendet: TAR2 liefert immer Bereichskennung 84 des
//Datenbausteins. P##evt_sec liefert 85 "Instanzdatenbaustein als
//Bereichskennung", was direkt die Instanzdaten adressiert.
      TAR2  ; // aktueller Instanzdaten-Pointer absolut
      UD    DW#16#FFFFFF; // Speicherbereich (84 "DB") ausblenden
      L     P##rARRAY; // relativer Pointer auf ARRAY (OFFEST)
      +D    ;
      T     #ptrARRAY; // absoluter Pointer auf ARRAY
NETWORK
TITLE =

      U     #evtNewValues;
      R     #evtNewValues;

NETWORK
TITLE =RESET

      UN    #RESET;
      SPB   ne4;

      L     0;
      T     #CNT_SEC;
      T     #CNT_MIN;
      T     #dIDX; // Zaehlvariable Minuten

      L     0.000000e+000;
      L     #rVALUE;
      T     #memSum1min;

ne4:  NOP   0;
NETWORK
TITLE =Zählen
//Bei Sollwert erreicht wird erst beim nächsten Takt der Integralwert
//zurückgesetzt, somit kann mit dem IMPULS der aktuelle Integralwert
//für die weitere Verarbeitung noch zur Verfügung.
//
      U     #TAKT_1S;
      FP    #HM_FP_TAKT;
      SPB   CNT;
      SPA   ne3;

CNT:  L     #CNT_SEC;
      INC   1;
      T     #CNT_SEC;

      L     #rVALUE;
      L     #memSum1min;
      +R    ;
      T     #memSum1min;

      L     #CNT_SEC;
      L     60;
      >=I   ;
      SPB   calc;
      SPA   ne3;

calc: NOP   0;
      S     #evtNewValues;

      L     0; // Sekunden rücksetzen
      T     #CNT_SEC;

      L     #memSum1min;
      L     6.000000e+001;
      /R    ;
      T     #rAVG_1min;
      T     #tmp_rAVG;

      L     0.000000e+000; // 1-Minuten-Summe löschen
      T     #memSum1min;

      L     #ptrARRAY;
      L     #dIDX;
      SLD   5; // *32 wegen 4-Byte-Wert = 32 Bit (S7-Pointer sind Bit-Pointer)
      +D    ;
      LAR1  ;

      L     #tmp_rAVG; // letzten Minuten Mittelwert  in ARRAY schreiben
      T     D [AR1,P#0.0]; // rARRAY[dIDX] = tmp_rAVG
      T     #tmp_rSUM;

      L     #dIDX;
      T     #dJ;

      L     1; // Schleifenzähler
      T     #I; // For I=1 To 14 (zum akt. Wert noch 14 alte addieren)

LOOP: NOP   0;

      L     #dIDX;
      L     #I;
      ITD   ;
      -D    ;
      UD    DW#16#F; // 0..15 Umlaufend
      SLD   5; // *32 wegen 4-Byte-Wert = 32 Bit (S7-Pointer sind Bit-Pointer)
      L     #ptrARRAY;
      +D    ;
      LAR1  ;

      L     D [AR1,P#0.0]; // rARRAY[dIDX-I] Überlauf berücksichtigt
      L     #tmp_rSUM;
      +R    ;
      T     #tmp_rSUM;

      L     #I;
      L     2; // 2 Werte wurden zum aktuellen addiert, d.h. Summe aus letzten 3 Minuten
      <>I   ;
      SPB   tst5;

      L     #tmp_rSUM;
      L     3.000000e+000;
      /R    ;
      T     #rAVG_3min;

tst5: L     #I;
      L     4; // 4 Werte wurden zum aktuellen addiert, d.h. Summe aus letzten 5 Minuten
      <>I   ;
      SPB   weit;

      L     #tmp_rSUM;
      L     5.000000e+000;
      /R    ;
      T     #rAVG_5min;

weit: L     #I; // Schleifenzähler
      +     1;
      T     #I;
      L     14;
      <I    ;
      SPB   LOOP; // LOOP IF I<14 (For I=1 To 14)

      L     #tmp_rSUM; // Summe über die letzten 15 Minuten
      L     1.500000e+001;
      /R    ;
      T     #rAVG_15min;

      L     #dIDX; // geschrieben wird in ARRAY[1..15] ARRAY[0] bleibt frei
      +     1;
      T     #dIDX;
      L     L#15;
      <D    ;
      SPB   ne3;
      L     L#0;
      T     #dIDX;
ne3:  NOP   0;
NETWORK
TITLE =FC-ENO-Ausgang = Zählimpuls
//
//
      L     #dIDX;
      T     #DSP_BUFFER_INDEX;

      SET   ;
      SAVE  ;
      CLR   ;
END_FUNCTION_BLOCK

FUNCTION_BLOCK "m7b_SpeedTakt"
TITLE =Antrieb Takten, wenn minSpeed unterschritten
//Anwendung: Frequenzumrichterantriebe ohne Fremdlüfter!
//           Antriebe ohne Fremdlüfter können nur auf etwa min 30Hz gefahren
//           werden. Soll weniger Drehzahl gefahren werden, dann muss mit
//           Puls/Pause getaktet werden. (z.B. Dosierschnecken)
//
//Dieser Baustein taktet unterhalb der MinDrehzahl mit dem Sollwert ensprechendem
//Puls/Pausenverhältnis. Als Sollwert wird dann der Minimalwert ausgegeben.
//
//z.B. 50Hz Motor bis 100Hz. d.h. 100Hz =100%
//     min Frequ: 30Hz
//
//d.h. bis 30% wird der Istwerteingang einfach druchgeschleift.
//bei Ist < 30% wird Sollwertausgang auf 30% eingefroren
//und der xTAKT Ausgang beginnt zu takten.
//
//bei 15% mit einem Taktverhältnis 50/50
//ist dann bei timeBase_100proz = 100sec, Puls=Pause=0.5 x timBase = 50sec
//
//Die untere %-Einstellung bei für Fmin berechnet man am besten mit
//FC103 "m7b_RPM_DRive"
//
//
//AUTOR: Stefan Maag, Dipl.-Ing. (FH) Elektrotechnik
//DATUM: 8/2018
//
//
//AENDERUNGSVERMERKE:
//--------------------------------------------------------------------------------
//DATUM        NAME        AENDERUNG
//--------------------------------------------------------------------------------
//
//--------------------------------------------------------------------------------
//
//HINWEISE:
AUTHOR : 'S.Maag'
FAMILY : Maagic7
VERSION : 0.1


VAR_INPUT
  FRG_Takten : BOOL ;	//Freigabe: 1: Takten wird bei unterschreiten von iMin aktiviert
  RESET : BOOL ;	//Reset
  iIST : INT ;	//Istwert
  iMin : INT ;	//Minimum
  timeBase_100proz : TIME ;	//Zeitbasis 100% (bei takten 50/50, Puls=Puase=0.5*timBase_100proz)
END_VAR
VAR_OUTPUT
  xTAKT : BOOL ;
  iSpeed : INT ;
  DSP_PULS : TIME ;
  DSP_PAUSE : TIME ;
END_VAR
VAR
  mi_MultiTimer : "m7b_MultiTimer";
  timPULS : TIME ;
  timPAUSE : TIME ;
END_VAR
VAR_TEMP
  CMD_TAKT : BOOL ;
  dTime : DINT ;
  d_ms_Puls : DINT ;
  dIST : DINT ;
  dMin : DINT ;
  Q_PulsPause : BOOL ;
  dTemp : DINT ;
  d_test : DINT ;
  DSP_Multi_T1 : TIME ;
  DSP_Multi_T2 : TIME ;
END_VAR
BEGIN
NETWORK
TITLE =



NETWORK
TITLE =Ist < Min => Takten
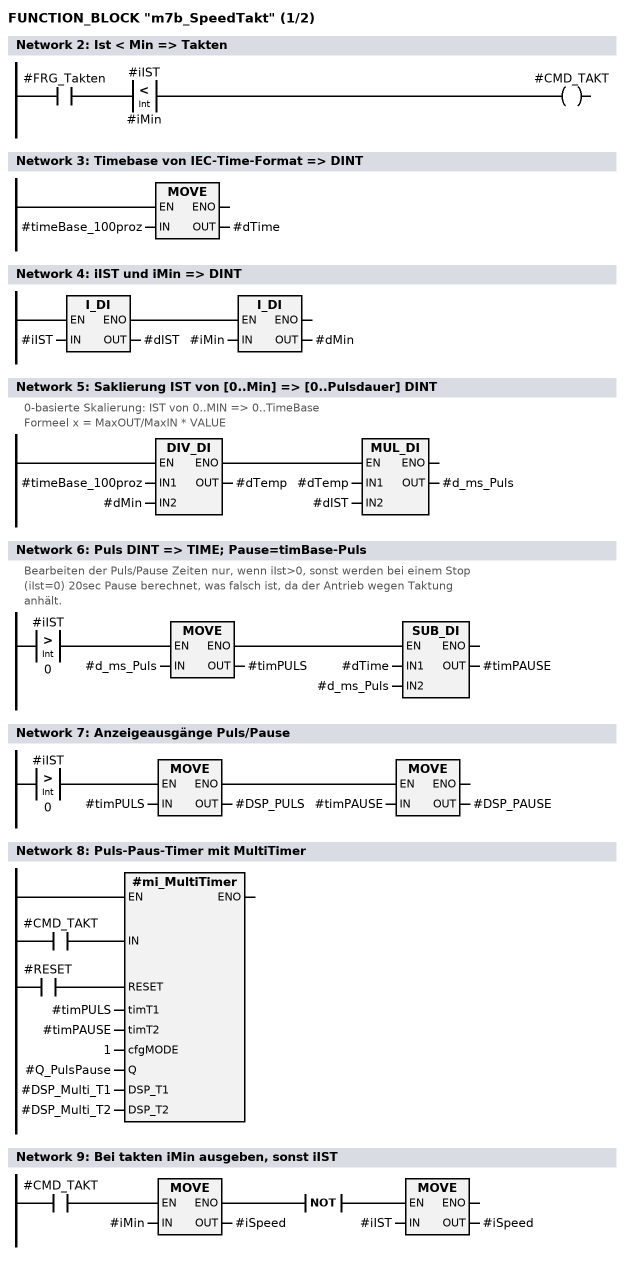

      U     #FRG_Takten;
      U(    ;
      L     #iIST;
      L     #iMin;
      <I    ;
      )     ;
      =     #CMD_TAKT;
NETWORK
TITLE =Timebase von IEC-Time-Format => DINT

      L     #timeBase_100proz;
      T     #dTime;
      NOP   0;
NETWORK
TITLE =iIST und iMin => DINT

      U(    ;
      L     #iIST;
      ITD   ;
      T     #dIST;


      SET   ;
      SAVE  ;
      CLR   ;
      U     BIE;
      )     ;
      SPBNB _001;
      L     #iMin;
      ITD   ;
      T     #dMin;
_001: NOP   0;
NETWORK
TITLE =Saklierung IST von [0..Min] => [0..Pulsdauer] DINT
//0-basierte Skalierung: IST von 0..MIN => 0..TimeBase
//
//Formeel x = MaxOUT/MaxIN * VALUE
      U(    ;
      L     #timeBase_100proz;
      L     #dMin;
      /D    ;
      T     #dTemp;
      UN    OV;
      SAVE  ;
      CLR   ;
      U     BIE;
      )     ;
      SPBNB _002;
      L     #dTemp;
      L     #dIST;
      *D    ;
      T     #d_ms_Puls;
_002: NOP   0;
NETWORK
TITLE =Puls DINT => TIME; Pause=timBase-Puls
//Bearbeiten der Puls/Pause Zeiten nur, wenn iIst>0, sonst werden bei einem Stop
//(iIst=0) 20sec Pause berechnet, was falsch ist, da der Antrieb wegen Taktung
//anhält.
      U(    ;
      U(    ;
      L     #iIST;
      L     0;
      >I    ;
      )     ;
      SPBNB _003;
      L     #d_ms_Puls;
      T     #timPULS;
      SET   ;
      SAVE  ;
      CLR   ;
_003: U     BIE;
      )     ;
      SPBNB _004;
      L     #dTime;
      L     #d_ms_Puls;
      -D    ;
      T     #timPAUSE;
_004: NOP   0;
NETWORK
TITLE =Anzeigeausgänge Puls/Pause

      U(    ;
      U(    ;
      L     #iIST;
      L     0;
      >I    ;
      )     ;
      SPBNB _005;
      L     #timPULS;
      T     #DSP_PULS;
      SET   ;
      SAVE  ;
      CLR   ;
_005: U     BIE;
      )     ;
      SPBNB _006;
      L     #timPAUSE;
      T     #DSP_PAUSE;
_006: NOP   0;
NETWORK
TITLE =Puls-Paus-Timer mit MultiTimer

      U     #CMD_TAKT;
      =     L     36.0;
      BLD   103;
      U     #RESET;
      =     L     36.1;
      BLD   103;
      CALL #mi_MultiTimer (
           IN                       := L     36.0,
           RESET                    := L     36.1,
           timT1                    := #timPULS,
           timT2                    := #timPAUSE,
           cfgMODE                  := 1,
           Q                        := #Q_PulsPause,
           DSP_T1                   := #DSP_Multi_T1,
           DSP_T2                   := #DSP_Multi_T2);
      NOP   0;
NETWORK
TITLE =Bei takten iMin ausgeben, sonst iIST

      U(    ;
      U     #CMD_TAKT;
      SPBNB _007;
      L     #iMin;
      T     #iSpeed;
      SET   ;
      SAVE  ;
      CLR   ;
_007: U     BIE;
      )     ;
      NOT   ;
      SPBNB _008;
      L     #iIST;
      T     #iSpeed;
_008: NOP   0;
NETWORK
TITLE =Taktausgang
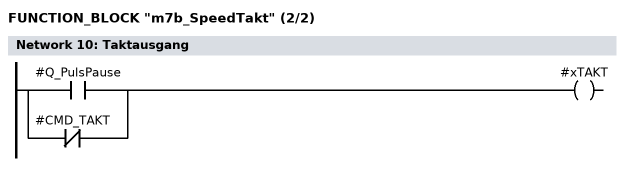

      O     #Q_PulsPause;
      ON    #CMD_TAKT;
      =     #xTAKT;
NETWORK
TITLE =FB-ENO = TAKT

      U     #xTAKT;
      SAVE  ;
END_FUNCTION_BLOCK

FUNCTION_BLOCK "Zwangsumschaltung"
TITLE =Systemumschaltung
//Umschaltung zwischen 2 redundanten Systemen. Z.B. 2 Pumpen, wobei 1 System
//immer als Ersatz vorhanden ist. Zwangsumschaltung 1x täglich nach Zeit
FAMILY : 'S.Maag'
VERSION : 0.1


VAR_INPUT
  IN_START : BOOL ;
  READY_1 : BOOL ;
  READY_2 : BOOL ;
  HOUR_1to2 : INT ;
  MIN_1to2 : INT ;
  HOUR_2to1 : INT ;
  MIN_2to1 : INT ;
  timOVERLAP : TIME ;	//Überlappungzeit bei Umschaltung
END_VAR
VAR_OUTPUT
  OUT_START_1 : BOOL ;
  OUT_START_2 : BOOL ;
END_VAR
VAR
  HM : BOOL ;
  SWTCH_to_2 : BOOL ;
  EVENT : BOOL ;
  OVERLAP : BOOL ;
  Q_TON_OVERLAP : BOOL ;
  TON_OVERLAP : "TON";
END_VAR
VAR_TEMP
  DATE_TIME : DATE_AND_TIME ;
  RET_VAL_READ_CLK : INT ;
  m_STD : INT ;
  m_MIN : INT ;
  HM_Q_TON_OVERLAP : BOOL ;
END_VAR
BEGIN
NETWORK
TITLE =



NETWORK
TITLE =Zeit in temporäreren Variablenbereich einlesen

      CALL "READ_CLK" (
           RET_VAL                  := #RET_VAL_READ_CLK,
           CDT                      := #DATE_TIME);
      NOP   0;
NETWORK
TITLE =Stunden, Minuten und Sekunden aus DATE_AND_TIME extrahieren
//Das DATE_AND_TIME Format benötigt 8 Byte im BCD-Format
//Der Wertebereich geht von DT#1990-1-1-0:0:0.0 bis DT#2089-12-31-23:59:59.999
//
//BYTE 0:  Jahr
//BYTE 1:  Monat
//BYTE 2:  Tag
//BYTE 3:  Stunde
//BYTE 4:  Minute
//BYTE 5:  Sekunde
//BYTE 6:  100er und 10er Stelle von Millisekunden
//BYTE 7:  Bit 4..7: 1er  Stelle von Millisekunden
//BYTE 7:  Bit 0..3: Wochentag (1=Sonntag, 2=Montag, ..., 7=Samstag)
      L     P##DATE_TIME;
      LAR1  ;

      L     B [AR1,P#3.0]; // Stunde
      BTI   ;
      T     #m_STD;

      L     B [AR1,P#4.0]; // Minute
      BTI   ;
      T     #m_MIN;

// Zeit prüfen und Event erzeugen
      L     #HOUR_1to2;
      L     #m_STD;
      <>I   ; // Stunde stimmt nicht, dann Ende
      SPB   END;

      L     #MIN_1to2;
      L     #m_MIN;
      <>I   ; // Minute stimmt nicht
      R     #HM; // HM wieder löschen
      SPB   END;

      U     #HM;
      SPB   END;
      S     #HM;
      S     #EVENT;

      UN    #SWTCH_to_2;
      =     #SWTCH_to_2;

END:  NOP   0;


NETWORK
TITLE =Zeit Überlappung mit Durchschaltung bei T:=0ms
//Sonderbehandlung IEC-Zeit, da Zeit mit T:=0 nicht anläuft
      U(    ;
      U     #EVENT;
      =     L     15.0;
      BLD   103;
      CALL #TON_OVERLAP (
           IN                       := L     15.0,
           PT                       := #timOVERLAP,
           Q                        := #HM_Q_TON_OVERLAP);

      U     BIE;
      )     ;
      U     #HM_Q_TON_OVERLAP;
      O     ;
      U     #EVENT;
      U(    ;
      L     #timOVERLAP;
      L     T#0MS;
      ==D   ;
      )     ;
      =     #Q_TON_OVERLAP;
      R     #EVENT;
NETWORK
TITLE =Overlap
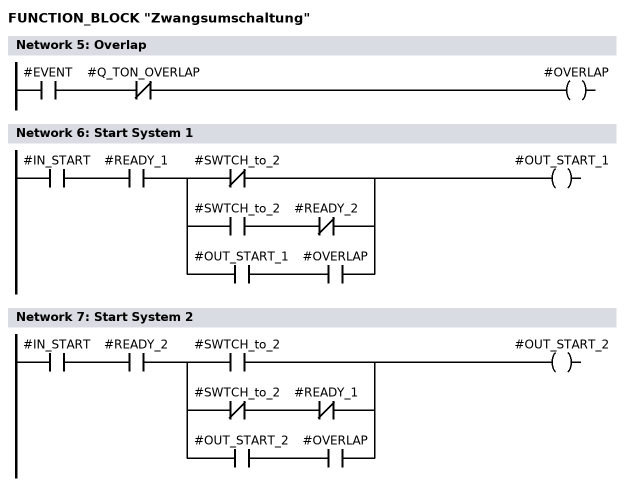

      U     #EVENT;
      UN    #Q_TON_OVERLAP;
      =     #OVERLAP;
NETWORK
TITLE =Start System 1



      U     #IN_START;
      U     #READY_1;
      U(    ;
      ON    #SWTCH_to_2;
      O     ;
      U     #SWTCH_to_2;
      UN    #READY_2;
      O     ;
      U     #OUT_START_1;
      U     #OVERLAP;
      )     ;
      =     #OUT_START_1;
NETWORK
TITLE =Start System 2

      U     #IN_START;
      U     #READY_2;
      U(    ;
      O     #SWTCH_to_2;
      O     ;
      UN    #SWTCH_to_2;
      UN    #READY_1;
      O     ;
      U     #OUT_START_2;
      U     #OVERLAP;
      )     ;
      =     #OUT_START_2;
END_FUNCTION_BLOCK

FUNCTION_BLOCK "cLevelMeter"
TITLE =Stufenschalter für 4 Geräte
AUTHOR : 'S.Maag'
VERSION : 0.1


VAR_INPUT
  rSOLL : REAL ;
  rS1_OFF : REAL ;
  rS1_ON : REAL ;
  rS2_OFF : REAL ;
  rS2_ON : REAL ;
  rS3_OFF : REAL ;
  rS3_ON : REAL ;
  rS4_OFF : REAL ;
  rS4_ON : REAL ;
END_VAR
VAR_OUTPUT
  Q1 : BOOL ;	//Device 1
  Q2 : BOOL ;	//Device 2
  Q3 : BOOL ;	//Device 3
  Q4 : BOOL ;	//Device 4
END_VAR
BEGIN
NETWORK
TITLE =



NETWORK
TITLE =Stufe 1: Hystereseschalter
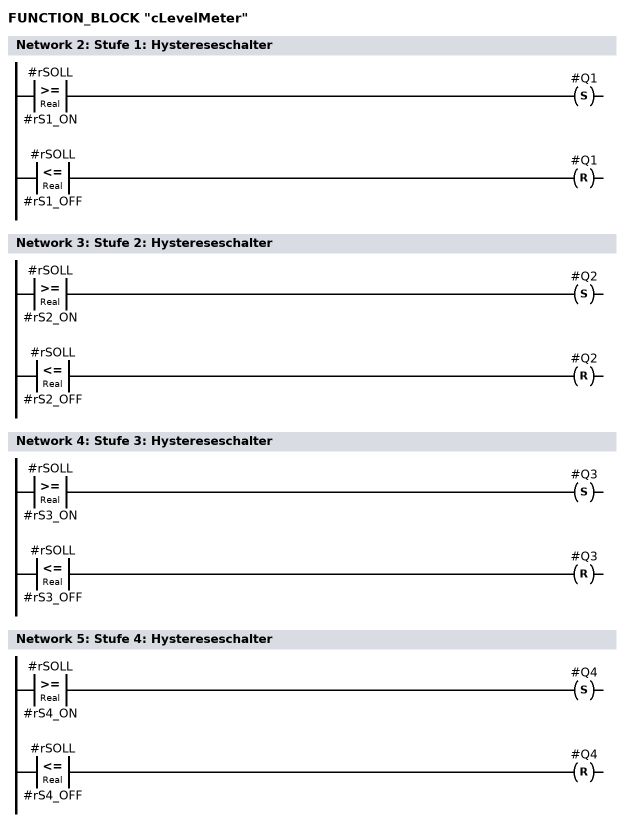

      U(    ;
      L     #rSOLL;
      L     #rS1_ON;
      >=R   ;
      )     ;
      S     #Q1;
      U(    ;
      L     #rSOLL;
      L     #rS1_OFF;
      <=R   ;
      )     ;
      R     #Q1;
      NOP   0;
NETWORK
TITLE =Stufe 2: Hystereseschalter

      U(    ;
      L     #rSOLL;
      L     #rS2_ON;
      >=R   ;
      )     ;
      S     #Q2;
      U(    ;
      L     #rSOLL;
      L     #rS2_OFF;
      <=R   ;
      )     ;
      R     #Q2;
      NOP   0;
NETWORK
TITLE =Stufe 3: Hystereseschalter

      U(    ;
      L     #rSOLL;
      L     #rS3_ON;
      >=R   ;
      )     ;
      S     #Q3;
      U(    ;
      L     #rSOLL;
      L     #rS3_OFF;
      <=R   ;
      )     ;
      R     #Q3;
      NOP   0;
NETWORK
TITLE =Stufe 4: Hystereseschalter

      U(    ;
      L     #rSOLL;
      L     #rS4_ON;
      >=R   ;
      )     ;
      S     #Q4;
      U(    ;
      L     #rSOLL;
      L     #rS4_OFF;
      <=R   ;
      )     ;
      R     #Q4;
      NOP   0;
END_FUNCTION_BLOCK

(*$PDIAG <?xml version='1.0' encoding='UTF-8'?>
<PDIAGDATA>
<Unit Block="FB1136" Type="14" Num="1136" TypeBType="0" TypeBNum="0">
<At id="1001">"m7b_ZylSensorCtrl"</At>
<At id="1003">19.09.2008 11:40:15</At>
<At id="1004">10.12.2020 20:10:02</At>
<At id="6109D">FB1136</At>
<At id="8006109D">FB1136</At>
</Unit>
</PDIAGDATA> *)
